// TwinCAT 3 PLC project LeakTesters
// ProgramVersion: 3.1.4024.0
// libraries:
//   Tc2_Standard, * (Beckhoff Automation GmbH)
//   Tc2_System, * (Beckhoff Automation GmbH)
//   Tc2_Utilities, * (Beckhoff Automation GmbH)
//   Tc3_EventLogger, * (Beckhoff Automation GmbH)
//   Tc3_Module, * (Beckhoff Automation GmbH)
//   VisuUserMgmt, * (System)
// project tree:
//   DUTs/ E_MachineState.TcDUT, E_StationState.TcDUT, ST_ActiveEventsHMI.TcDUT (not stored), ST_AlarmHistory.TcDUT (not stored), ST_Events.TcDUT, ST_Heightlimit.TcDUT, ST_MachineStatusStruct.TcDUT, ST_MasterControlStruct.TcDUT, ST_MeasureStatistics.TcDUT, ST_Nest.TcDUT, ST_PartsInspection.TcDUT, ST_StandardStationStruct.TcDUT, ST_UserLogHMI.TcDUT (not stored)
//   DUTs/IO/i28/ st_i28General_I_O.TcDUT (not stored), st_i28LasResult.TcDUT (not stored), st_i28LiveMeasurement.TcDUT (not stored)
//   DUTs/IO/ E_BoxDiag.TcDUT, E_BoxState.TcDUT, E_TerminalState.TcDUT, st_Box_Info.TcDUT, st_EL1809.TcDUT, st_EL2809.TcDUT, st_Terminal_Info.TcDUT
//   GVLs/ GVL_Constants.TcGVL, GVL_HMI_GLOBAL.TcGVL, GVL_IO.TcGVL, GVL_MASTER.TcGVL, GVL_PERSIST.TcGVL
//   / PlcTask.TcTTO
//   POUs/A_Master/ Main_Master.TcPOU, PRG_FaultHandling.TcPOU, PRG_MachineStatus.TcPOU, PRG_MasterCycle.TcPOU, PRG_MasterSystemTime.TcPOU, PRG_TerminBoxInfo.TcPOU
//   POUs/C_LeakTest/ PRG_Fault_LeakTest.TcPOU, PRG_LeakTest.TcPOU, PRG_LeakTestEvents_Info.TcPOU
//   POUs/E_HMI/ PRG_HMI.TcPOU
//   POUs/G_Utility/ FB_Alarms.TcPOU, FB_BoxInfo.TcPOU, FB_DayOfYear.TcPOU, FB_EventLog.TcPOU (not stored), FB_HeightMeasurement.TcPOU, FB_HeightTest.TcPOU, FB_Pulse.TcPOU (not stored), FB_TerminalInfo.TcPOU, FB_TimeControl.TcPOU (not stored), PRG_Puls.TcPOU
//   POUs/ MAIN.TcPOU
// real-time tasks:
//   TASK PlcTask: cycle T#10ms, priority 20, ADS port 350
// I/O:
//   DEVICE Device 1 (EtherCAT), AmsNetId 172.18.236.47.2.1
//     Term 9 (EK1100) [EK1100 EtherCAT Coupler (2A E-Bus)]
//       Term 10 (EL6070-0033) [EL6070-0033 1Ch. Licence key terminal, individual licences]
//       Term 11 (EL1809) [EL1809 16Ch. Dig. Input 24V, 3ms]
//       Term 12 (EL2809-0015) [EL2809-0015 16Ch. Dig. Output 24V DC, 0.35A, not short-circuit proof]
//       Term 13 (EL6631) [EL6631 PROFINET IO Controller]
//       Term 14 (EL9011) [EL9011 End Terminal]
//   DEVICE Device 2 (EL6631), AmsNetId 172.18.236.47.3.1
//     i28 [Cincinnati Test Systems 1-port Device 00210]
//       modules: Term 10 (DAP Module), Term 11 (PLC Input), Term 12 (PLC Output  )
// variable links:
//   LeakTesters/LeakTesters Instance <-> Device 1 (EtherCAT)/Term 9 (EK1100)/Term 11 (EL1809)
//     PlcTask Inputs/GVL_IO.dwTerminalInfo[3].nTerminal_State <-> InfoData/State
//     PlcTask Inputs/GVL_IO.dw_T02_EL1809.iCalmpClosed <-> Channel 1/Input
//     PlcTask Inputs/GVL_IO.dw_T02_EL1809.iPartPresent <-> Channel 2/Input
//   LeakTesters/LeakTesters Instance <-> Device 1 (EtherCAT)/Term 9 (EK1100)/Term 12 (EL2809-0015)
//     PlcTask Inputs/GVL_IO.dwTerminalInfo[4].nTerminal_State <-> InfoData/State
//     PlcTask Outputs/GVL_IO.dw_T03_EL2809.qEL2809_Ch3 <-> Channel 3/Output
//     PlcTask Outputs/GVL_IO.dw_T03_EL2809.qPassIndicatorGreen <-> Channel 1/Output
//     PlcTask Outputs/GVL_IO.dw_T03_EL2809.qRejectIndicatorRed <-> Channel 2/Output
//   LeakTesters/LeakTesters Instance <-> Device 1 (EtherCAT)/Term 9 (EK1100)/Term 13 (EL6631)
//     PlcTask Inputs/GVL_IO.dwTerminalInfo[5].nTerminal_State <-> InfoData/State
//   LeakTesters/LeakTesters Instance <-> Device 2 (EL6631)/i28
//     PlcTask Inputs/GVL_IO.dwBoxInfo[16].nPnIoBoxDiag <-> Inputs/PnIoBoxDiag
//     PlcTask Inputs/GVL_IO.dwBoxInfo[16].nPnIoBoxState <-> Inputs/PnIoBoxState
//     PlcTask Inputs/GVL_IO.dw_B07_i28General_I_O.bInput1 <-> API/Term 11 (PLC Input)/Subterm 15 (Instrument Status)/Inputs/Instrument Status/User_Configurable_Input_1
//     PlcTask Inputs/GVL_IO.dw_B07_i28General_I_O.bInput10 <-> API/Term 11 (PLC Input)/Subterm 15 (Instrument Status)/Inputs/Instrument Status/User_Configurable_Input_10
//     PlcTask Inputs/GVL_IO.dw_B07_i28General_I_O.bInput11 <-> API/Term 11 (PLC Input)/Subterm 15 (Instrument Status)/Inputs/Instrument Status/User_Configurable_Input_11
//     PlcTask Inputs/GVL_IO.dw_B07_i28General_I_O.bInput12 <-> API/Term 11 (PLC Input)/Subterm 15 (Instrument Status)/Inputs/Instrument Status/User_Configurable_Input_12
//     PlcTask Inputs/GVL_IO.dw_B07_i28General_I_O.bInput13 <-> API/Term 11 (PLC Input)/Subterm 15 (Instrument Status)/Inputs/Instrument Status/User_Configurable_Input_13
//     PlcTask Inputs/GVL_IO.dw_B07_i28General_I_O.bInput14 <-> API/Term 11 (PLC Input)/Subterm 15 (Instrument Status)/Inputs/Instrument Status/User_Configurable_Input_14
//     PlcTask Inputs/GVL_IO.dw_B07_i28General_I_O.bInput15 <-> API/Term 11 (PLC Input)/Subterm 15 (Instrument Status)/Inputs/Instrument Status/User_Configurable_Input_15
//     PlcTask Inputs/GVL_IO.dw_B07_i28General_I_O.bInput16 <-> API/Term 11 (PLC Input)/Subterm 15 (Instrument Status)/Inputs/Instrument Status/User_Configurable_Input_16
//     PlcTask Inputs/GVL_IO.dw_B07_i28General_I_O.bInput2 <-> API/Term 11 (PLC Input)/Subterm 15 (Instrument Status)/Inputs/Instrument Status/User_Configurable_Input_2
//     PlcTask Inputs/GVL_IO.dw_B07_i28General_I_O.bInput3 <-> API/Term 11 (PLC Input)/Subterm 15 (Instrument Status)/Inputs/Instrument Status/User_Configurable_Input_3
//     PlcTask Inputs/GVL_IO.dw_B07_i28General_I_O.bInput4 <-> API/Term 11 (PLC Input)/Subterm 15 (Instrument Status)/Inputs/Instrument Status/User_Configurable_Input_4
//     PlcTask Inputs/GVL_IO.dw_B07_i28General_I_O.bInput5 <-> API/Term 11 (PLC Input)/Subterm 15 (Instrument Status)/Inputs/Instrument Status/User_Configurable_Input_5
//     PlcTask Inputs/GVL_IO.dw_B07_i28General_I_O.bInput6 <-> API/Term 11 (PLC Input)/Subterm 15 (Instrument Status)/Inputs/Instrument Status/User_Configurable_Input_6
//     PlcTask Inputs/GVL_IO.dw_B07_i28General_I_O.bInput7 <-> API/Term 11 (PLC Input)/Subterm 15 (Instrument Status)/Inputs/Instrument Status/User_Configurable_Input_7
//     PlcTask Inputs/GVL_IO.dw_B07_i28General_I_O.bInput8 <-> API/Term 11 (PLC Input)/Subterm 15 (Instrument Status)/Inputs/Instrument Status/User_Configurable_Input_8
//     PlcTask Inputs/GVL_IO.dw_B07_i28General_I_O.bInput9 <-> API/Term 11 (PLC Input)/Subterm 15 (Instrument Status)/Inputs/Instrument Status/User_Configurable_Input_9
//     PlcTask Inputs/GVL_IO.dw_B07_i28General_I_O.bInstrumentReady <-> API/Term 11 (PLC Input)/Subterm 15 (Instrument Status)/Inputs/Instrument Status/Instrument_Ready
//     PlcTask Inputs/GVL_IO.dw_B07_i28General_I_O.bMalfunction <-> API/Term 11 (PLC Input)/Subterm 15 (Instrument Status)/Inputs/Instrument Status/Malfunction
//     PlcTask Inputs/GVL_IO.dw_B07_i28General_I_O.bProgramAccept <-> API/Term 11 (PLC Input)/Subterm 15 (Instrument Status)/Inputs/Instrument Status/Program_Accept
//     PlcTask Inputs/GVL_IO.dw_B07_i28General_I_O.bProgramReject <-> API/Term 11 (PLC Input)/Subterm 15 (Instrument Status)/Inputs/Instrument Status/Program_Reject
//     PlcTask Inputs/GVL_IO.dw_B07_i28General_I_O.bTestActiveLiveData <-> API/Term 11 (PLC Input)/Subterm 15 (Instrument Status)/Inputs/Instrument Status/Test_Active_Live_Data
//     PlcTask Inputs/GVL_IO.dw_B07_i28General_I_O.nCurrentProgramNumber <-> API/Term 11 (PLC Input)/Subterm 15 (Instrument Status)/Inputs/Current_Program Number
//     PlcTask Inputs/GVL_IO.dw_B07_i28LastResult.ibTestEvaluation0 <-> API/Term 11 (PLC Input)/Subterm 17 (Last test result)/Inputs/Test Evaluation Code/Test_Evaluation_Code_Bit_0
//     PlcTask Inputs/GVL_IO.dw_B07_i28LastResult.ibTestEvaluation1 <-> API/Term 11 (PLC Input)/Subterm 17 (Last test result)/Inputs/Test Evaluation Code/Test_Evaluation_Code_Bit_1
//     PlcTask Inputs/GVL_IO.dw_B07_i28LastResult.ibTestEvaluation2 <-> API/Term 11 (PLC Input)/Subterm 17 (Last test result)/Inputs/Test Evaluation Code/Test_Evaluation_Code_Bit_2
//     PlcTask Inputs/GVL_IO.dw_B07_i28LastResult.ibTestEvaluation3 <-> API/Term 11 (PLC Input)/Subterm 17 (Last test result)/Inputs/Test Evaluation Code/Test_Evaluation_Code_Bit_3
//     PlcTask Inputs/GVL_IO.dw_B07_i28LastResult.inChannelNumber <-> API/Term 11 (PLC Input)/Subterm 17 (Last test result)/Inputs/Channel Number
//     PlcTask Inputs/GVL_IO.dw_B07_i28LastResult.inMeasurement1 <-> API/Term 11 (PLC Input)/Subterm 17 (Last test result)/Inputs/Result Measurement 1
//     PlcTask Inputs/GVL_IO.dw_B07_i28LastResult.inMeasurement2 <-> API/Term 11 (PLC Input)/Subterm 17 (Last test result)/Inputs/Result Measurement 2
//     PlcTask Inputs/GVL_IO.dw_B07_i28LastResult.inPartEvaluation <-> API/Term 11 (PLC Input)/Subterm 17 (Last test result)/Inputs/Part Evaluation Code
//     PlcTask Inputs/GVL_IO.dw_B07_i28LastResult.inPrecisionCode <-> API/Term 11 (PLC Input)/Subterm 17 (Last test result)/Inputs/Precision Code
//     PlcTask Inputs/GVL_IO.dw_B07_i28LastResult.inProgramNumber <-> API/Term 11 (PLC Input)/Subterm 17 (Last test result)/Inputs/Program Number
//     PlcTask Inputs/GVL_IO.dw_B07_i28LastResult.inTestPort <-> API/Term 11 (PLC Input)/Subterm 17 (Last test result)/Inputs/Test Port
//     PlcTask Inputs/GVL_IO.dw_B07_i28LastResult.inTestType <-> API/Term 11 (PLC Input)/Subterm 17 (Last test result)/Inputs/Test Type Code
//     PlcTask Inputs/GVL_IO.dw_B07_i28LastResult.inUniqueID <-> API/Term 11 (PLC Input)/Subterm 17 (Last test result)/Inputs/Unique ID
//     PlcTask Inputs/GVL_IO.dw_B07_i28LastResult.inUnitCode1 <-> API/Term 11 (PLC Input)/Subterm 17 (Last test result)/Inputs/Unit Code[0]
//     PlcTask Inputs/GVL_IO.dw_B07_i28LastResult.inUnitCode2 <-> API/Term 11 (PLC Input)/Subterm 17 (Last test result)/Inputs/Unit Code[1]
//     PlcTask Inputs/GVL_IO.dw_B07_i28LastResult.inVariableCode1 <-> API/Term 11 (PLC Input)/Subterm 17 (Last test result)/Inputs/Variable Code[0]
//     PlcTask Inputs/GVL_IO.dw_B07_i28LastResult.inVariableCode2 <-> API/Term 11 (PLC Input)/Subterm 17 (Last test result)/Inputs/Variable Code[1]
//     PlcTask Inputs/GVL_IO.dw_B07_i28LiveMeasurement.inCurrentProgramNumber <-> API/Term 11 (PLC Input)/Subterm 16 (Live Measurement Data)/Inputs/Current Program Number
//     PlcTask Inputs/GVL_IO.dw_B07_i28LiveMeasurement.inMeasurement1 <-> API/Term 11 (PLC Input)/Subterm 16 (Live Measurement Data)/Inputs/Measurement 1 (Timer)
//     PlcTask Inputs/GVL_IO.dw_B07_i28LiveMeasurement.inMeasurement2 <-> API/Term 11 (PLC Input)/Subterm 16 (Live Measurement Data)/Inputs/Measurement 2 (Pressure)
//     PlcTask Inputs/GVL_IO.dw_B07_i28LiveMeasurement.inMeasurement3 <-> API/Term 11 (PLC Input)/Subterm 16 (Live Measurement Data)/Inputs/Measurement 3 (Pressure Loss/Rate)
//     PlcTask Inputs/GVL_IO.dw_B07_i28LiveMeasurement.inMeasurement4 <-> API/Term 11 (PLC Input)/Subterm 16 (Live Measurement Data)/Inputs/Measurement 4 (Flow/Leak)
//     PlcTask Inputs/GVL_IO.dw_B07_i28LiveMeasurement.inPrecisionCode1 <-> API/Term 11 (PLC Input)/Subterm 16 (Live Measurement Data)/Inputs/Precision Code[0]
//     PlcTask Inputs/GVL_IO.dw_B07_i28LiveMeasurement.inPrecisionCode2 <-> API/Term 11 (PLC Input)/Subterm 16 (Live Measurement Data)/Inputs/Precision Code[1]
//     PlcTask Inputs/GVL_IO.dw_B07_i28LiveMeasurement.inPrecisionCode3 <-> API/Term 11 (PLC Input)/Subterm 16 (Live Measurement Data)/Inputs/Precision Code[2]
//     PlcTask Inputs/GVL_IO.dw_B07_i28LiveMeasurement.inPrecisionCode4 <-> API/Term 11 (PLC Input)/Subterm 16 (Live Measurement Data)/Inputs/Precision Code[3]
//     PlcTask Inputs/GVL_IO.dw_B07_i28LiveMeasurement.inSegmentCode <-> API/Term 11 (PLC Input)/Subterm 16 (Live Measurement Data)/Inputs/Segment Code
//     PlcTask Inputs/GVL_IO.dw_B07_i28LiveMeasurement.inUniqueID <-> API/Term 11 (PLC Input)/Subterm 16 (Live Measurement Data)/Inputs/Unique ID
//     PlcTask Inputs/GVL_IO.dw_B07_i28LiveMeasurement.inUnitCode1 <-> API/Term 11 (PLC Input)/Subterm 16 (Live Measurement Data)/Inputs/Unit Code[0]
//     PlcTask Inputs/GVL_IO.dw_B07_i28LiveMeasurement.inUnitCode2 <-> API/Term 11 (PLC Input)/Subterm 16 (Live Measurement Data)/Inputs/Unit Code[1]
//     PlcTask Inputs/GVL_IO.dw_B07_i28LiveMeasurement.inUnitCode3 <-> API/Term 11 (PLC Input)/Subterm 16 (Live Measurement Data)/Inputs/Unit Code[2]
//     PlcTask Inputs/GVL_IO.dw_B07_i28LiveMeasurement.inUnitCode4 <-> API/Term 11 (PLC Input)/Subterm 16 (Live Measurement Data)/Inputs/Unit Code[3]
//     PlcTask Inputs/GVL_IO.dw_B07_i28LiveMeasurement.inVariableCode1 <-> API/Term 11 (PLC Input)/Subterm 16 (Live Measurement Data)/Inputs/Variable Code[0]
//     PlcTask Inputs/GVL_IO.dw_B07_i28LiveMeasurement.inVariableCode2 <-> API/Term 11 (PLC Input)/Subterm 16 (Live Measurement Data)/Inputs/Variable Code[1]
//     PlcTask Inputs/GVL_IO.dw_B07_i28LiveMeasurement.inVariableCode3 <-> API/Term 11 (PLC Input)/Subterm 16 (Live Measurement Data)/Inputs/Variable Code[2]
//     PlcTask Inputs/GVL_IO.dw_B07_i28LiveMeasurement.inVariableCode4 <-> API/Term 11 (PLC Input)/Subterm 16 (Live Measurement Data)/Inputs/Variable Code[3]
//     PlcTask Outputs/GVL_IO.dw_B07_i28General_I_O.bChangeProgram <-> API/Term 12 (PLC Output  )/Subterm 18 (Instrument Control )/Outputs/Instrument Control/Change_Program
//     PlcTask Outputs/GVL_IO.dw_B07_i28General_I_O.bOutput1 <-> API/Term 12 (PLC Output  )/Subterm 18 (Instrument Control )/Outputs/Instrument Control/User_Configurable_Output_1
//     PlcTask Outputs/GVL_IO.dw_B07_i28General_I_O.bOutput10 <-> API/Term 12 (PLC Output  )/Subterm 18 (Instrument Control )/Outputs/Instrument Control/User_Configurable_Output_10
//     PlcTask Outputs/GVL_IO.dw_B07_i28General_I_O.bOutput11 <-> API/Term 12 (PLC Output  )/Subterm 18 (Instrument Control )/Outputs/Instrument Control/User_Configurable_Output_11
//     PlcTask Outputs/GVL_IO.dw_B07_i28General_I_O.bOutput12 <-> API/Term 12 (PLC Output  )/Subterm 18 (Instrument Control )/Outputs/Instrument Control/User_Configurable_Output_12
//     PlcTask Outputs/GVL_IO.dw_B07_i28General_I_O.bOutput13 <-> API/Term 12 (PLC Output  )/Subterm 18 (Instrument Control )/Outputs/Instrument Control/User_Configurable_Output_13
//     PlcTask Outputs/GVL_IO.dw_B07_i28General_I_O.bOutput14 <-> API/Term 12 (PLC Output  )/Subterm 18 (Instrument Control )/Outputs/Instrument Control/User_Configurable_Output_14
//     PlcTask Outputs/GVL_IO.dw_B07_i28General_I_O.bOutput15 <-> API/Term 12 (PLC Output  )/Subterm 18 (Instrument Control )/Outputs/Instrument Control/User_Configurable_Output_15
//     PlcTask Outputs/GVL_IO.dw_B07_i28General_I_O.bOutput16 <-> API/Term 12 (PLC Output  )/Subterm 18 (Instrument Control )/Outputs/Instrument Control/User_Configurable_Output_16
//     PlcTask Outputs/GVL_IO.dw_B07_i28General_I_O.bOutput2 <-> API/Term 12 (PLC Output  )/Subterm 18 (Instrument Control )/Outputs/Instrument Control/User_Configurable_Output_2
//     PlcTask Outputs/GVL_IO.dw_B07_i28General_I_O.bOutput3 <-> API/Term 12 (PLC Output  )/Subterm 18 (Instrument Control )/Outputs/Instrument Control/User_Configurable_Output_3
//     PlcTask Outputs/GVL_IO.dw_B07_i28General_I_O.bOutput4 <-> API/Term 12 (PLC Output  )/Subterm 18 (Instrument Control )/Outputs/Instrument Control/User_Configurable_Output_4
//     PlcTask Outputs/GVL_IO.dw_B07_i28General_I_O.bOutput5 <-> API/Term 12 (PLC Output  )/Subterm 18 (Instrument Control )/Outputs/Instrument Control/User_Configurable_Output_5
//     PlcTask Outputs/GVL_IO.dw_B07_i28General_I_O.bOutput6 <-> API/Term 12 (PLC Output  )/Subterm 18 (Instrument Control )/Outputs/Instrument Control/User_Configurable_Output_6
//     PlcTask Outputs/GVL_IO.dw_B07_i28General_I_O.bOutput7 <-> API/Term 12 (PLC Output  )/Subterm 18 (Instrument Control )/Outputs/Instrument Control/User_Configurable_Output_7
//     PlcTask Outputs/GVL_IO.dw_B07_i28General_I_O.bOutput8 <-> API/Term 12 (PLC Output  )/Subterm 18 (Instrument Control )/Outputs/Instrument Control/User_Configurable_Output_8
//     PlcTask Outputs/GVL_IO.dw_B07_i28General_I_O.bOutput9 <-> API/Term 12 (PLC Output  )/Subterm 18 (Instrument Control )/Outputs/Instrument Control/User_Configurable_Output_9
//     PlcTask Outputs/GVL_IO.dw_B07_i28General_I_O.bReset <-> API/Term 12 (PLC Output  )/Subterm 18 (Instrument Control )/Outputs/Instrument Control/Reset
//     PlcTask Outputs/GVL_IO.dw_B07_i28General_I_O.bSetProgram[0] <-> API/Term 12 (PLC Output  )/Subterm 18 (Instrument Control )/Outputs/Desired Program Number[0]
//     PlcTask Outputs/GVL_IO.dw_B07_i28General_I_O.bSetProgram[1] <-> API/Term 12 (PLC Output  )/Subterm 18 (Instrument Control )/Outputs/Desired Program Number[1]
//     PlcTask Outputs/GVL_IO.dw_B07_i28General_I_O.bSetProgram[2] <-> API/Term 12 (PLC Output  )/Subterm 18 (Instrument Control )/Outputs/Desired Program Number[2]
//     PlcTask Outputs/GVL_IO.dw_B07_i28General_I_O.bSetProgram[3] <-> API/Term 12 (PLC Output  )/Subterm 18 (Instrument Control )/Outputs/Desired Program Number[3]
//     PlcTask Outputs/GVL_IO.dw_B07_i28General_I_O.bSetProgram[4] <-> API/Term 12 (PLC Output  )/Subterm 18 (Instrument Control )/Outputs/Desired Program Number[4]
//     PlcTask Outputs/GVL_IO.dw_B07_i28General_I_O.bSetProgram[5] <-> API/Term 12 (PLC Output  )/Subterm 18 (Instrument Control )/Outputs/Desired Program Number[5]
//     PlcTask Outputs/GVL_IO.dw_B07_i28General_I_O.bSetProgram[6] <-> API/Term 12 (PLC Output  )/Subterm 18 (Instrument Control )/Outputs/Desired Program Number[6]
//     PlcTask Outputs/GVL_IO.dw_B07_i28General_I_O.bSetProgram[7] <-> API/Term 12 (PLC Output  )/Subterm 18 (Instrument Control )/Outputs/Desired Program Number[7]
//     PlcTask Outputs/GVL_IO.dw_B07_i28General_I_O.bStart <-> API/Term 12 (PLC Output  )/Subterm 18 (Instrument Control )/Outputs/Instrument Control/Start
//     PlcTask Outputs/GVL_IO.dw_B07_i28General_I_O.bStop <-> API/Term 12 (PLC Output  )/Subterm 18 (Instrument Control )/Outputs/Instrument Control/Stop
//     PlcTask Outputs/GVL_IO.dw_B07_i28General_I_O.bVentHalt <-> API/Term 12 (PLC Output  )/Subterm 18 (Instrument Control )/Outputs/Instrument Control/Vent_Halt

CONFIGURATION LeakTesters
    RESOURCE PLC ON TwinCAT3
        TASK PlcTask(INTERVAL := T#10ms, PRIORITY := 20);
        PROGRAM MAIN WITH PlcTask : MAIN;
    END_RESOURCE
END_CONFIGURATION

// ---- DUTs/E_MachineState.TcDUT
{attribute 'qualified_only'}
{attribute 'strict'}
TYPE E_MachineState :
(
	SYSTEM_POWER_UP:=0,
	IMMEDIATE_STOPPED:=100,
	SYSTEM_INITIALISING:=110,
	SYSTEM_READY_TO_START:=120,
	SYSTEM_AUTO_CYCLE:=130,
	SYSTEM_DWELL:=140,
	STOPPING:=145,
	CYCLE_STOPPED:=150,
	MANUAL_MODE:=160 ,
	MAINTENANCE_MODE:=165,
	IMMEDIATE_FAULT:=170,
	CYCLE_STOP_FAULT:=180
);
END_TYPE

// ---- DUTs/E_StationState.TcDUT
{attribute 'qualified_only'}
{attribute 'strict'}
TYPE E_StationState :
(
	RESETTING := 0,
	PRE_ELIMINARY_CHECKS,
	TRY_HOMING,
	HOMING,
	HOMING_DONE,
	READY,
	STARTING,
	DWELL,
	OPERATING,
	
//VALUES FOR UCB
	
//standard steps
	ERROR,
	COMPLETE
);
END_TYPE

// ---- DUTs/IO/E_BoxDiag.TcDUT
{attribute 'qualified_only'}
{attribute 'strict'}
TYPE E_BoxDiag :
(
	No_diagnosis                                   :=0,
    IOC_AR_is_not_established                      := 1,
    IOC_AR_is_established                          := 2,
    IOC_AR_is_established_but_no_application_ready := 4,
    IOC_AR_is_established_but_module_difference    := 8,
    At_least_one_AlarmCR_got_a_diagnosis_alarm     := 10,
    At_least_one_InputCR_is_invalid                := 100,
    At_least_one_InputCR_Provider_is_in_stop       := 200,
    At_least_one_InputCR_Problemindicator_is_set   := 400,
    At_least_one_OutputCR_is_invalid               := 1000,
    At_least_one_OutputCR_Provider_is_in_stop      := 2000,
    At_least_one_OutputCR_Problemindicator_is_set  := 4000
);
END_TYPE

// ---- DUTs/IO/E_BoxState.TcDUT
{attribute 'qualified_only'}
{attribute 'strict'}
TYPE E_BoxState :
(
	No_error                                                                     := 0,
    Profinet_device_state_machine_is_in_boot_mode                                := 1,
    Device_NOT_found                                                             := 2,
    The_stationname_is_not_unique                                                := 3,
    IP_could_not_be_set                                                          := 4,
    IP_conflict                                                                  := 5,
    DCP_set_was_not_successful                                                   := 6,
    Watchdog_error                                                               := 7,
    Datahold_error                                                               := 8,
    RTC3_Sync_mode_could_NOT_be_initiated                                        := 9,
    Profinet_controller_has_a_link_error                                         := 10,
    The_aliasname_is_not_unique                                                  := 11,
    The_automatic_name_assignement_isnt_possible_wrong_device_type               := 12,
    IOC_AR_is_established_but_no_application_ready                               := 13,
    IOC_AR_is_established_but_module_difference                                  := 14,
    At_least_one_InputCR_is_invalid_provider_in_stop_OR_problemindicator_is_set  := 15,
    At_least_one_OutputCR_is_invalid_provider_in_stop_OR_problemindicator_is_set := 16,
    Only_for_EtherCAT_gateways_WC_State_OF_cyclic_EtherCAT_frame_is_1            := 31
);
END_TYPE

// ---- DUTs/IO/E_TerminalState.TcDUT
{attribute 'qualified_only'}
{attribute 'strict'}
TYPE E_TerminalState :
(
	 INIT   := 0 ,
     PREOP  := 2 ,
     BOOT   := 3 ,
     SAFEOP := 4 ,
     OP     := 8 

);
END_TYPE

// ---- DUTs/IO/st_Box_Info.TcDUT
TYPE st_Box_Info :
STRUCT
	nPnIoBoxState    AT%I* : UINT;
    nPnIoBoxDiag     AT%I* : UINT;
    eBoxState              : E_BoxState;
	eBoxDiag               : E_BoxDiag;
	fbBoxInfo              : FB_BoxInfo;
	sBoxState              : STRING;
	sBoxDiag               : STRING;
	
END_STRUCT
END_TYPE

// ---- DUTs/IO/st_EL1809.TcDUT
TYPE st_EL1809 :
STRUCT
	
		//--------------------------------------------------------------------------------------------------------
	sTerminalName                                           :   STRING(200):= 'EL1809 | 16-Channel Digital Input';
    //============================================================================================================================	
	// TERMINAL - EL1809 16-Channel Digital Input Terminal 
    (*Terminal 02*)
	iCalmpClosed                			AT %I*			: 	BOOL;	// EL1809 channel 1
	iPartPresent                            AT %I*			: 	BOOL;	// EL1809 channel 2
	iEL1809_Ch3								AT %I*	 		: 	BOOL;	// EL1809 channel 3
	iEL1809_Ch4								AT %I*	 		: 	BOOL;	// EL1809 channel 4
	iEL1809_Ch5	    		                AT %I*	 		: 	BOOL;	// EL1809 channel 5 		     			
	iEL1809_Ch6			  					AT %I*			: 	BOOL;	// EL1809 channel 6
	iEL1809_Ch7		    					AT %I*	 		: 	BOOL;	// EL1809 channel 7 
	iEL1809_Ch8			   					AT %I*	 		: 	BOOL;	// EL1809 channel 8 
    iEL1809_Ch9			                    AT %I*	 		: 	BOOL;	// EL1809 channel 9 
	iEL1809_Ch10			                AT %I*          :   BOOL;   // EL1809 channel 10 
	iEL1809_Ch11		                    AT %I*          :   BOOL;   // EL1809 channel 11
	iEL1809_Ch12		                    AT %I*          :   BOOL;   // EL1809 channel 12	   
	iEL1809_Ch13			   		    	AT %I*	 		: 	BOOL;	// EL1809 channel 13   
	iEL1809_Ch14							AT %I*	 		: 	BOOL;	// EL1809 channel 14 
	iEL1809_Ch15	  						AT %I*			: 	BOOL;	// EL1809 channel 15  
	iEL1809_Ch16							AT %I*	 		: 	BOOL;	// EL1809 channel 16  

END_STRUCT
END_TYPE

// ---- DUTs/IO/st_EL2809.TcDUT
TYPE st_EL2809 :
STRUCT
	
		sTerminalName                                           :   STRING(200):= 'EL2809 | 16-Channel Digital Output';
	//=============================================================================================================
	// TERMINAL - EL2809	16-Channel Digital Output Terminal	 (Term ...)
	qPassIndicatorGreen 					AT %Q*			: 	BOOL;	// EL2809 channel 1
	qRejectIndicatorRed						AT %Q* 			: 	BOOL;	// EL2809 channel 2
	qEL2809_Ch3				                AT %Q*          :   BOOL;   // EL2809 channel 3
	qEL2809_Ch4				            	AT %Q*          :   BOOL;   // EL2809 channel 4   	
	qEL2809_Ch5		     					AT %Q*	 		: 	BOOL;	// EL2809 channel 5	
	qEL2809_Ch6	    		            	AT %Q*	 		: 	BOOL;	// EL2809 channel 6	
    qEL2809_Ch7	                        	AT %Q*          :   BOOL;   // EL2809 channel 7	
	qEL2809_Ch8								AT %Q*	 		: 	BOOL;	// EL2809 channel 8 
	qEL2809_Ch9				                AT %Q*          :   BOOL;   // EL2809 channel 9
	qEL2809_Ch10				            AT %Q*          :   BOOL;   // EL2809 channel 10   	
	qEL2809_Ch11		     				AT %Q*	 		: 	BOOL;	// EL2809 channel 11	
	qEL2809_Ch12	    		            AT %Q*	 		: 	BOOL;	// EL2809 channel 12	
    qEL2809_Ch13	                        AT %Q*          :   BOOL;   // EL2809 channel 13	
	qEL2809_Ch14							AT %Q*	 		: 	BOOL;	// EL2809 channel 14 
    qEL2809_Ch15        			        AT %Q*	 		: 	BOOL;	// EL2809 channel 15 
	qEL2809_Ch16                            AT %Q*	 		: 	BOOL;	// EL2809 channel 16 
	
	
END_STRUCT
END_TYPE

// ---- DUTs/IO/st_Terminal_Info.TcDUT
TYPE st_Terminal_Info :
STRUCT
	nTerminal_State                        AT %I*			:    UINT;	// Terminal State from IO Terminal Info Data
    eTerminal_State                                         :    E_TerminalState;
	sTerminalInfo                                           :    STRING;
    fbTerminalInfo                                          :    FB_TerminalInfo;
END_STRUCT
END_TYPE

// ---- DUTs/ST_Events.TcDUT
TYPE ST_Events :
STRUCT
	bImmediateFault				:BOOL;
	bCycleStopFault				:BOOL;
	bCycleStopRequest			:BOOL;

	bEventTextsSet				:BOOL; //True after event texts are set 
	aEventFlags					:ARRAY[0..127] OF BOOL;
	aEventTimers				:ARRAY[0..127] OF TON;
	aEventTexts					:ARRAY[0..127] OF T_MaxString;
END_STRUCT
END_TYPE

// ---- DUTs/ST_Heightlimit.TcDUT
TYPE ST_Heightlimit :
STRUCT
	LOW:   INT;
	HIGH:  INT;
	
END_STRUCT
END_TYPE

// ---- DUTs/ST_MachineStatusStruct.TcDUT
TYPE ST_MachineStatusStruct :
STRUCT
	nState						: INT;
	//nStateBuffer				: INT;
	eMachineState				:E_MachineState;	
	bSystemPowerUp 				:BOOL;
	bImmediateStopped 			:BOOL;
	bSystemInitialising 		:BOOL;
	bSystemReadyToStart 		:BOOL;
	bSystemAutoCycle 			:BOOL;
	bSystemDwell 				:BOOL;
	bSystemStopping				:BOOL;	
	bCycleStopped 				:BOOL;
	bImmediateFault 			:BOOL;
	bCycleStopFault 			:BOOL;
	bManualMode					:BOOL;
    bSystemStandby              :BOOL;		
	
	sMachineStatusText			:STRING;
	nMachineStatusTxtCol		:DWORD;
	nMachineStatusColour		:DWORD;
	sBannerTextColor			:STRING ;
	sBannerBckColor				:STRING ;
END_STRUCT
END_TYPE

// ---- DUTs/ST_MasterControlStruct.TcDUT
TYPE ST_MasterControlStruct :
STRUCT
	bAbort									:BOOL;
	bNoMachineImmediateFault				:BOOL;
	bNoStationImmediateFault				:BOOL;
	bNoCycleStopFault						:BOOL;
	bAllStationsHomed						:BOOL;
	bAllStationsCycledStopped				:BOOL;
	bCycleStopRequest						:BOOL;
	bDwellRequest							:BOOL;
	bManualModeRequest						:BOOL;
	bFreezeMachineStatus					:BOOL;
	bPowerUpTimerComplete					:BOOL;
	bSystemInitialisingTimerComplete		:BOOL;
	bSystemInitialisingTimeoutComplete		:BOOL;
	bResetImmediateFaultDelay				:BOOL;
	
	bAllStationsSafeToIndex					:BOOL;
	bAllStationsOKToIndex					:BOOL;
	bAllStationsNotMoving					:BOOL;
	
	bLineClearanceRequest					:BOOL;
	bLineClearanceComplete					:BOOL;
END_STRUCT
END_TYPE

// ---- DUTs/ST_MeasureStatistics.TcDUT
TYPE ST_MeasureStatistics :
STRUCT
	 bOutLimitMax	 : BOOL;
	 bOutLimitMin    : BOOL;
	 nMesureFaultMin : UINT;
	 nMesureFaultMax : UINT;
END_STRUCT
END_TYPE

// ---- DUTs/ST_Nest.TcDUT
TYPE ST_Nest :
STRUCT
		 

	 
     bNestPartProced    : BOOL;
	 bNestPresent       : BOOL;
	 
	 bPiecePass			: BOOL;
	 bPieceReject		: BOOL;
	 bLeakPass			: BOOL;
	 bLeakReject		: BOOL;
	 
	 
	 sLeakHMI			: WSTRING;
	 sPieceHMI			: WSTRING;

	 
	 sDate				: STRING;
	 sTime				: STRING;

END_STRUCT
END_TYPE

// ---- DUTs/ST_PartsInspection.TcDUT
TYPE ST_PartsInspection :
STRUCT
	
	nPartsGood						: DINT;
	nTotalPartsGood					: DINT;
	nPartsFailed					: DINT;
	nTotalPartsFailed				: DINT;					
	
	bPartok							: BOOL;
	bPartFail						: BOOL;
END_STRUCT
END_TYPE

// ---- DUTs/ST_StandardStationStruct.TcDUT
TYPE ST_StandardStationStruct :
STRUCT
	
		// Station Manager => Master Control
	nState 							: 	DINT := 100;//Station Cycle State
	bStationWaitOnInit              :   BOOL;       //Station Waiting For Initialisation Request
	bStationWaitOnRequest			:	BOOL;		//Station In Valide State Avaiting For Request Command
	bStationInProgress				: 	BOOL;		//Station In Progress With Cycle
	bStationInProgressInit          :   BOOL;       //Station In Progress With Imotialisation     
	bStationComplete				: 	BOOL;		//Station Complete Cycle - Flag Set After Every Cycle Finsh
	bStationCycleStopped			: 	BOOL;
	bStationHomed					: 	BOOL;		//Station Homed - All Station Functions Are Homed 
	bStationDone					:	BOOL;		//Sequence Finished With Success - Flag Set For One PLC Cycle
	bStationNotMoving				: 	BOOL;		//Station Parts Are Not Moving
	bStationInDwell					: 	BOOL;		//Station Waiting For External Action By Operator
	bStationAcknowledge             :   BOOL;       //Station Acknowledge request from Master 
	bStationInitDone                :   BOOL;       //Station Initialisation Progress Done
	// Master Control => Station Manager
	bStationInitRequest             :   BOOL;       //Request Commnad To Start Station Initialisation
	bStationRequest					: 	BOOL;		//Request Commnad To Start Station Cycle
	bStationCompleteAck				: 	BOOL;		//Request Commnad To Start Station Cycle
	bStationHomingRequest			:	BOOL;		//Staion Homing Requested By Manager Or Internal Functions
	bStationAbort					: 	BOOL;		//Station Abort By Manager
	bNoCycleStopRequest				:	BOOL;		//Stop Cycle Requested By Manager
	bNoCycleStopFault				: 	BOOL;		//No  Stop Fault On Station - Immidiat STOP Station
	bNoImmediateFault				: 	BOOL;		//No Immediate Fault On Station - Immidiat STOP Machine
	
	
	bStationManualRequestHMI		:	BOOL;		//Sequence Cycle Requested From HMI
	bStationInManualMode			:	BOOL;		//Station Sequence Manage By Operator

	bStationInStandByMode			:	BOOL;		//Sequence In Stand By State
	bStationFreezedByManager		: 	BOOL;		//Sequence Cycle Freezed (Suspend)  By Manager
	
	eStationState					: 	E_StationState; // state of sequence
	
	bPartOK							:	BOOL;		// 1-Cycle succeed
	bPartReject                     :   BOOL;       // 1-Cycle failed

	
	bStationWaiting                 :   BOOL; // Station in the  positiont waiting for work done
	bStationCycleCondition          :   BOOL; // Station in cycle move
END_STRUCT
END_TYPE

// ---- GVLs/GVL_Constants.TcGVL
VAR_GLOBAL CONSTANT
	sWHITE                              :   STRING(40)  := '{"color":"rgba(255,255,255,255)"}';
    sBLACK                              :   STRING(40)  := '{"color":"rgba(0,0,0,1)"}';
    sYELLOW                             :   STRING(40)  := '{"color":"rgba(255,255,0,1)"}';
    sGREEN                             	:   STRING(40)  := '{"color":"rgba(70,166,63,1)"}';
	sLGREEN                             :   STRING(40)  := '{"color":"rgba(58,211,20,1)"}';
    sORANGE                             :   STRING(40)  := '{"color":"rgba(255,153,51,1)"}';
    sNYPROORANGE                        :   STRING(40)  := '{"color":"rgba(255,140,0,1)"}';
    sRED                                :   STRING(40)  := '{"color":"rgba(255,0,0,1)"}';
	sLRED                               :   STRING(40)  := '{"color":"rgba(233,53,44,1)"}';
    sBLUE                               :   STRING(40)  := '{"color":"rgba(0,0,255,1)"}';
	sLBLUE                              :   STRING(40)  := '{"color":"rgba(0,162,232,1)"}';
    sGREY                               :   STRING(40)  := '{"color":"rgba(164,158,158,1)"}';
    sScreenGREY                         :   STRING(40)  := '{"color":"rgba(225,225,225,1)"}';
    sDARKGREY                           :   STRING(40)  := '{"color":"rgba(50,50,50,1)"}';
    sPURPLE                             :   STRING(40)  := '{"color":"rgba(128,0,128,1)"}';
    sVIOLET                             :   STRING(40)  := '{"color":"rgba(204,153,255,1)"}';
    sTRANSP                             :   STRING(40)  := '{"color":"rgba(255,255,255,0)"}';
    sGREENPass                          :   STRING(40)  := '{"color":"rgba(0,153,51,1)"}';
    sREDFail                            :   STRING(40)  := '{"color":"rgba(244,68,68,255)"}';
    sBLUEInProgress                     :   STRING(40)  := '{"color":"rgba(54,100,221,1)"}';
	sGREENISHTEAColor					:	STRING(40)  := '{"color":"rgba(60,192,134,255)"}'	;		

	nBLACK								: 	DWORD 	:= 	16#FF000000;	 // format: TTRRGGBB where T -> 00 = full transparency and FF = full opaque
	nWHITE								: 	DWORD 	:= 	16#FFFFFFFF;
	nYELLOW								: 	DWORD 	:= 	16#FFFFFF00; 
	nGREEN								: 	DWORD 	:= 	16#FF008A00;
	nLIGHTGREEN                         :   DWORD   :=  16#FF98FB89;
	nORANGE								: 	DWORD 	:= 	16#FFFFA500;
	nNYPROORANGE						:	DWORD	:=	16#FFF05322;//F05322;
	nRED								: 	DWORD 	:= 	16#FFFF0000;
	nBLUE								: 	DWORD 	:= 	16#FF0000FF;
	nLIGHTBLUE                          :   DWORD   :=  16#FF08ADF4;//FF9FDDFB;
	nGREY								: 	DWORD 	:= 	16#FFA9A9A9;	
	nDARKGREY							:	DWORD	:=	16#FF808080;
	nPURPLE								:	DWORD	:=	16#FF800080;
	nVIOLET								:	DWORD	:=	16#FFEE82EE;
	nTRANSP								:	DWORD	:=	16#00FFFFFF;	// full transparent WHITE
	
	nLCColNormal						:	DWORD	:= 16#10008A00;		// light curtain green
	nLCColBroken						:	DWORD	:= 16#64FF0000;		// light curtain red
END_VAR

// ---- GVLs/GVL_HMI_GLOBAL.TcGVL
{attribute 'qualified_only'}
VAR_GLOBAL
	
	//User Log, Shut down, Quit HMI
	bQuitHmi						: BOOL;
	sUserGroup						: STRING;
	sUserGroup2						: STRING;
	sUserName						: STRING;
	bLogOut							: BOOL;
	bUserLogedIntSignal				: BOOL;
	bShutDown						: BOOL;
	
	
	
	
	
	//General
	bStopButton						: BOOL;
	bStartButton					: BOOL;
	bResetButton					: BOOL;
	nRegionMain						: INT;
	bTrigerCamMan					: BOOL;
	bResetGoodParts					: BOOL;
	bResetFailedParts				: BOOL;
	bManualModeOff					: ARRAY[1..2] OF BOOL;
	
	aEventTexts						: ARRAY [0..767] OF T_MaxSTring; //Event texts - set only once
	bEventTextsSet					: BOOL;
	aEventFlags						: ARRAY [0..767] OF BOOL;		//All event states combined from master na stations
	aActiveEvents					: ARRAY [0..39] OF T_MaxSTring;	//Active events - connected to Alarm scree in HMI	
	stActiveEventsHMI				: ARRAY [0..39] OF ST_ActiveEventsHMI;
	
	aStatistics						: ARRAY [1..201] OF ST_Nest; // **LA 04092025 >> : ARRAY [1..200] OF ST_Nest;
	sMessageToOperator				: WSTRING(200);
	sActualProcess					: WSTRING(200);
	aIOScreen						: ARRAY [0..8] OF STRING(200);
	aManualScreen					: ARRAY [0..2] OF STRING(200);
	bResetPassAndFail				: BOOL;
	bEnableManualMode				: BOOL;
	bRejectPieceAcknowledge			: BOOL;
	bRejectPieceDialogTrig			: BOOL;
	bAutoCycleFaultDialog			: BOOL;
	bStopperPressEnable				: BOOL;
	nGeneralCycTime					: DINT;
		
	
	// ------ Screen Info / Data -----------	
	sSystemDate					: STRING;
	sSystemTime					: STRING;
	ntAMSNetID					: T_AmsNetId := '172.18.236.47.1.1';
	sStopperEnableDisable		:STRING(30); 
	
	
	//Leak Tester
	bLeakTestPass					: BOOL;
	uSetLeakProgramID				: USINT;
	bSetLeakProgramID				: BOOL;
	bResetLeakMan					: BOOL;
	bStartLeakMan					: BOOL;
	bStopLeakMan					: BOOL;
	bLoadLeakProg					: BOOL;
	uNewLeakProgID					: USINT;
		
	bResetLeakGoodParts				: BOOL;
	bResetLeakBadParts				: BOOL;
	nLeakTestCycTime				: DINT;	

END_VAR
VAR_GLOBAL PERSISTENT
	stAlarmHistory				:ARRAY [00..250] OF ST_AlarmHistory;
	aEventLog					:ARRAY [0..250] OF T_MaxSTring;	//Event log - connected to alarm history in HMI	
	aTimeLog					:ARRAY [0..250] OF T_MaxSTring;
	aDateLog					:ARRAY [0..250] OF T_MaxSTring;			
END_VAR

// ---- GVLs/GVL_IO.TcGVL
{attribute 'qualified_only'}
VAR_GLOBAL
	
    //--------------------------------------------------------------------------------------------------------

    dwTerminalInfo                                          : ARRAY[0..20] OF  st_Terminal_Info; // all terminal's status information 
	dwBoxInfo                                               : ARRAY[15..17] OF st_Box_Info;//Camera, Leak, Height
	//--------------------------------------------------------------------------------------------------------
	
	(* Terminal *)
	
	//	dw_T01_EK1100                                                	| EtherCAT Coupler 
	//	dw_T02_EL6070-0033                                           	| EtherCAT Terminal, license key for TwinCAT 3.1
	
	dw_T02_EL1809                                                		: st_EL1809; //16 Channel Digital Input ( 24VDC ) 
	dw_T03_EL2809                                                		: st_EL2809; // 16 Channel Digital Output ( 24VDC )
	//dw_T04_EL6631                                                	| EtherCAT Terminal, 2-port communication interface, PROFINET RT, controller - Data for Box's MDU1020 and SR2000W
 	//  dw_T05_EL9011                                                	| Bus end cover for E-bus contacts
	
	dw_B07_i28General_I_O												: st_i28General_I_O;
	dw_B07_i28LastResult												: st_i28LasResult;
	dw_B07_i28LiveMeasurement											: st_i28LiveMeasurement;
	
	
	
END_VAR

// ---- GVLs/GVL_MASTER.TcGVL
{attribute 'qualified_only'}
VAR_GLOBAL
	(*-----------------------------------------------------------------------------------------------------------------*)
	// System Pulses 
	bFlash1Hz						: BOOL;
	bFlash2Hz						: BOOL;
	bFlash4Hz				   		: BOOL;
	bFlash10Hz						: BOOL;
	bFlash10BHz        		  		: BOOL;
	bFlash100Hz      	      		: BOOL;
	bFlashScale       	      		: BOOL;
	bFlashScale4       		  		: BOOL;
	bFlashScale5        	  		: BOOL;
	bFlashingFreq2			  		: BOOL;
	bFlashScaleFast       	  		: BOOL;
	
//Master Control
	stMachineStatus					: ST_MachineStatusStruct;	
	stMasterControl					: ST_MasterControlStruct;
  	stStationSruct                  : ARRAY[0..1] OF ST_StandardStationStruct; (* Station 0 - Master
                                                                                  Station 1 - Leak test                                                           
                                                                                   *)

	
																				   
	stNest							: ST_Nest;                                                                        
	stAlarms                        : ARRAY [0..1] OF ST_Events;
	
	bManualModeTrigger				: BOOL;
	bFirstScan				:   BOOL;
	tFirstScan				:   TON;



	
																				   

END_VAR

// ---- GVLs/GVL_PERSIST.TcGVL
{attribute 'qualified_only'}
VAR_GLOBAL PERSISTENT
	
stPartsInspection			: ST_PartsInspection;
stUserLogHMI				: ARRAY[0..250] OF ST_UserLogHMI;
UserId						: UINT;
ast_i28LasResult            : ARRAY [0..250] OF st_i28LasResult;
nLeakTestID					: UINT;

nCycleNumber				: INT;
	
END_VAR

// ---- POUs/MAIN.TcPOU
PROGRAM MAIN
VAR
END_VAR

Main_Master();

END_PROGRAM

// ---- POUs/A_Master/Main_Master.TcPOU
PROGRAM Main_Master
VAR
	i                       :INT; //Int to handle user log index	
	k						:INT; //Int to handle user log index
	j						:INT;
	l						:INT;
	
	//////UserLog
	
	sUserGroupID			:	STRING;
	nSize					:	UDINT					:=9;
	nLen					:	UDINT					:=18;
	npos					:	UDINT					:=1;
	tonUserLogOut           :	Tc2_Standard.TON;
	fbStringFormatter       :	Tc2_Utilities.FB_FormatString;
	fbEventLogger			:	FB_EventLog;
	rUserLoggedIn			: 	R_TRIG;
	tUserLoggedIn			: 	TON;
	bFirstScan				:   BOOL;
	tFirstScan				:   TON;

	bUserLoggedIn			: 	BOOL;
	

	
	
	/////ShutDown&Quit
	closeChrome 			: 	NT_StartProcess;	
	ntShutdown					: TC2_Utilities.NT_Shutdown;
	ntError						: BOOL;
	ntBusy						: BOOL;
	ntErrorID					: UDINT;

	
	
	/////General

END_VAR

PRG_FaultHandling(aAlarms := GVL_Master.stAlarms );
PRG_Fault_LeakTest(aAlarms := GVL_Master.stAlarms);


PRG_MachineStatus();
PRG_MasterCycle(stStationStruct:= GVL_Master.stStationSruct[0]);
PRG_MasterSystemTime();
ACT_ShutdownAndQuit();
ACT_UserLog();
MapUnitEventsToHmi();
PRG_HMI();
PRG_Puls();
ACT_FirstScan();
PRG_TerminBoxInfo();

//gfggf




PRG_LeakTestEvents_Info();





//Stations
PRG_LeakTest(stStationStruct:= GVL_Master.stStationSruct[1]);




fbEventLogger(	bEnable       	:= PRG_MasterSystemTime.bReadyToRead AND GVL_MASTER.stMasterControl.bPowerUpTimerComplete,
			    sDateTime     	:= PRG_MasterSystemTime.sDateTimeSpaces,
			    aEventFlags   	:= GVL_HMI_GLOBAL.aEventFlags,
			    aEventTexts   	:= GVL_HMI_GLOBAL.aEventTexts,
			    aActiveEvents 	:= GVL_HMI_GLOBAL.aActiveEvents,
			    aEventLog     	:= GVL_HMI_GLOBAL.aEventLog,
				siDate			:= GVL_HMI_GLOBAL.sSystemDate,
				siTime			:= GVL_HMI_GLOBAL.sSystemTime,
				soDate			:= GVL_HMI_GLOBAL.aDateLog,
				soTime			:= GVL_HMI_GLOBAL.aTimeLog
);



 

IF GVL_MASTER.bFlashScale THEN
FOR j := 0 TO 39 DO
	
GVL_HMI_GLOBAL.stActiveEventsHMI[j].sActiveEvents := GVL_HMI_GLOBAL.aActiveEvents[j];
END_FOR
FOR l:=0 TO 250 DO
	
	GVL_HMI_GLOBAL.stAlarmHistory[l].sEventlog 	:= GVL_HMI_GLOBAL.aEventLog[l];
	GVL_HMI_GLOBAL.stAlarmHistory[l].sDate		:= GVL_HMI_GLOBAL.aDateLog[l];
	GVL_HMI_GLOBAL.stAlarmHistory[l].sTime		:= GVL_HMI_GLOBAL.aTimeLog[l];
END_FOR
ELSE 
	
j:=0; 
l:=0;

END_IF

ACTION ACT_FirstScan:
tFirstScan(IN := NOT bFirstScan, PT := T#5S);
END_ACTION

ACTION ACT_ShutdownAndQuit:
closeChrome(
    NetId := '',
    PathStr := 'C:\Windows\System32\mshta vbscript:Execute("CreateObject(""WScript.Shell"").Run ""powershell -c',
    DirName := 'C:\Windows\System32\WindowsPowerShell\v1.0',
    ComndLine := 'taskkill /F /IM chrome.exe /T"", 0: window.close")',
    Start := GVL_HMI_GLOBAL.bQuitHmi,
    TmOut := DEFAULT_ADS_TIMEOUT
);
 
GVL_HMI_GLOBAL.bQuitHmi:= FALSE;

ntShutdown(NETID := GVL_HMI_GLOBAL.ntAMSNetID, DELAY := 5, START := GVL_HMI_GLOBAL.bShutDown, BUSY => ntBusy, ERR => ntError, ERRID => ntErrorID);
END_ACTION

ACTION ACT_UserLog:

//Getting user group

Tc2_Utilities.DELETE2( ADR(GVL_HMI_GLOBAL.sUserGroup), ADR(sUserGroupID), NSize, Nlen, nPos) ;

IF sUserGroupID = 'Administ' THEN
	
	GVL_HMI_GLOBAL.sUserGroup2 := 'Administrator';

ELSE GVL_HMI_GLOBAL.sUserGroup2 := sUserGroupID;
	

END_IF


//Logout 

tonUserLogOut( IN := (sUserGroupID = 'Administ' OR sUserGroupID ='Engineer') AND GVL_HMI_GLOBAL.bUserLogedIntSignal , PT := T#10M);

IF tonUserLogOut.Q AND (sUserGroupID = 'Administ' OR sUserGroupID ='Engineer') THEN
	
	GVL_HMI_GLOBAL.bLogOut 	:= TRUE;

	ELSE GVL_HMI_GLOBAL.bLogOut := FALSE;

END_IF

tUserLoggedIn( IN := GVL_HMI_GLOBAL.bUserLogedIntSignal, PT := T#2S);

rUserLoggedIn( CLK := tUserLoggedIn.Q);


IF rUserLoggedIn.Q THEN
	
	FOR i :=200 TO 1 BY (-1) DO
		GVL_PERSIST.stUserLogHMI[i]	:= GVL_PERSIST.stUserLogHMI[i-1];
	END_FOR
	
	GVL_PERSIST.stUserLogHMI[0].UserLog := GVL_HMI_GLOBAL.sUserName;
	GVL_PERSIST.stUserLogHMI[0].UserLogTime := GVL_HMI_GLOBAL.sSystemTime;
	GVL_PERSIST.stUserLogHMI[0].UserLogDate := GVL_HMI_GLOBAL.sSystemDate;

END_IF
END_ACTION

METHOD MapUnitEventsToHMI : BOOL
VAR_INPUT
END_VAR

VAR
	i		:INT; 	//Unit index
	j		:INT;	//Unit event index
	k		:INT; 	//HMI event index	
END_VAR
//Set event texts first
IF GVL_Master.stAlarms[0].bEventTextsSet AND
   GVL_Master.stAlarms[1].bEventTextsSet AND
   NOT GVL_HMI_GLOBAL.bEventTextsSet 
THEN
	SetEventTexts();
		
	GVL_HMI_GLOBAL.bEventTextsSet := TRUE;
END_IF

//Map events from master and stations into HMI events
IF GVL_HMI_GLOBAL.bEventTextsSet THEN
	k := 0; 
	FOR i := 0 TO 4 DO
		FOR j := 0 TO 128 - 1 DO
			GVL_HMI_GLOBAL.aEventFlags[k] := GVL_Master.stAlarms[i].aEventFlags[j];
			k := k + 1;
		END_FOR
	END_FOR
END_IF
END_METHOD

METHOD SetEventTexts : BOOL
VAR_INPUT
END_VAR
VAR
	i				:INT; 	//Unit index
	j				:INT;	//HMI event index
	k				:INT;	//
END_VAR
//Set global event texts based on unit event texts (master and stations
k := 0;
FOR i := 0 TO 1 DO
	//For each unit (master, station1, station2)
	//Alarm texts
	FOR j := 0 TO 99 DO
		fbStringFormatter(	sFormat := 'Alarm No. %d - %s', 
					 	arg1 := F_INT(k), 
						arg2 := F_String(GVL_Master.stAlarms[i].aEventTexts[j]),
						sOut => GVL_HMI_GLOBAL.aEventTexts[k]);
						
		k := k + 1; //Increment global events index
	END_FOR
	
	//Messages
	FOR j := 100 TO 127 DO
		fbStringFormatter(	sFormat := 'Message No. %d - %s', 
					 		arg1 := F_INT(k), 
							arg2 := F_String(GVL_Master.stAlarms[i].aEventTexts[j]),
							sOut => GVL_HMI_GLOBAL.aEventTexts[k]);
							
		k := k + 1; //Increment global events index
	END_FOR
END_FOR
END_METHOD

END_PROGRAM

// ---- POUs/A_Master/PRG_FaultHandling.TcPOU
PROGRAM PRG_FaultHandling
VAR
	
	i							: INT;
	bFlagResetOn				: BOOL;
	bStationCycleFaultFlag		: BOOL;




END_VAR
VAR_IN_OUT

  aAlarms  : ARRAY[0..1] OF ST_Events;
END_VAR

ACT_FaultTrig();

(************************************** Faults reset **********************************************)
IF   GVL_HMI_GLOBAL.bResetButton THEN 
	FOR i := 0 TO 127 DO
		GVL_MASTER.stAlarms[0].aEventFlags[i] := FALSE;
	END_FOR
END_IF


//===============================================================
//Initialize event texts on first scan
IF NOT GVL_MASTER.stAlarms[0].bEventTextsSet THEN
	SetEventTexts();
	GVL_MASTER.stAlarms[0].bEventTextsSet := TRUE;
END_IF
IF NOT GVL_MASTER.stAlarms[0].bEventTextsSet THEN
	GVL_MASTER.stAlarms[0].bEventTextsSet := FALSE;
END_IF


(***************************************************************************************************)
//Immediate fault
GVL_MASTER.stAlarms[0].bImmediateFault := FALSE;
FOR i := 0 TO 32DO
	GVL_MASTER.stAlarms[0].bImmediateFault := GVL_MASTER.stAlarms[0].bImmediateFault OR GVL_MASTER.stAlarms[0].aEventFlags[i];
END_FOR

//Cycle stop fault
GVL_MASTER.stAlarms[0].bCycleStopFault := FALSE;
FOR i := 33 TO 79 DO
	GVL_MASTER.stAlarms[0].bCycleStopFault := GVL_MASTER.stAlarms[0].bCycleStopFault OR GVL_MASTER.stAlarms[0].aEventFlags[i];
END_FOR

//Cycle stop request
GVL_MASTER.stAlarms[0].bCycleStopRequest := FALSE;
FOR i := 80 TO 99 DO
	GVL_MASTER.stAlarms[0].bCycleStopRequest := GVL_MASTER.stAlarms[0].bCycleStopRequest OR GVL_MASTER.stAlarms[0].aEventFlags[i];
END_FOR


(**************************** Master Fault Monitors ***********************************************)
(* Station Immediate Fault Monitor *)
GVL_MASTER.stMasterControl.bNoStationImmediateFault := 	NOT GVL_MASTER.stAlarms[0].bImmediateFault AND NOT GVL_MASTER.stAlarms[1].bImmediateFault;

(**************************************************************************************************)
(**************************** Cycle stop falt  **************************************)
bStationCycleFaultFlag := NOT GVL_MASTER.stAlarms[0].bCycleStopFault AND NOT GVL_MASTER.stAlarms[1].bCycleStopFault;

(**************************** Master Immediate Fault Monitor **************************************)
GVL_MASTER.stMasterControl.bNoMachineImmediateFault := NOT GVL_MASTER.stAlarms[0].bImmediateFault AND NOT GVL_MASTER.stAlarms[1].bImmediateFault;

									
(**************************************************************************************************)

(* Master Cycle Stop Fault Monitor *)
GVL_MASTER.stMasterControl.bNoCycleStopFault := NOT GVL_MASTER.stAlarms[0].bCycleStopFault;

ACTION ACT_FaultTrig:
(**************************************************************************************************)
(**************************** Master Immediate Fault Stop *****************************************)
(**************************************************************************************************)

//Beckhoff EL1809 Not Operational
IF NOT GVL_MASTER.stMachineStatus.bSystemPowerUp AND GVL_IO.dwTerminalInfo[3].nTerminal_State<>8 THEN
	GVL_MASTER.stAlarms[0].aEventFlags[33] := TRUE;
END_IF
//Beckhoff EL2809 Not Operational
IF NOT GVL_MASTER.stMachineStatus.bSystemPowerUp AND GVL_IO.dwTerminalInfo[4].nTerminal_State<>8 THEN
	GVL_MASTER.stAlarms[0].aEventFlags[34] := TRUE;
END_IF

//System stopping timeout
GVL_MASTER.stAlarms[0].aEventTimers[38](IN := ( GVL_MASTER.stMachineStatus.bSystemStopping ), PT := T#20S);
IF GVL_MASTER.stAlarms[0].aEventTimers[38].Q THEN
	GVL_MASTER.stAlarms[0].aEventFlags[38] := TRUE;	
END_IF
//User not Log In
GVL_MASTER.stAlarms[0].aEventTimers[39](IN := (GVL_HMI_GLOBAL.sUserName=''), PT := T#40MS);
IF GVL_MASTER.stAlarms[0].aEventTimers[39].Q THEN
	GVL_MASTER.stAlarms[0].aEventFlags[39] := TRUE;	
END_IF
//User LOG-Off Timeout Manual Mode
GVL_MASTER.stAlarms[0].aEventTimers[40](IN:= ((GVL_HMI_GLOBAL.sUserName='') AND GVL_MASTER.stMachineStatus.bManualMode),PT:= T#1S); 
IF GVL_MASTER.stAlarms[0].aEventTimers[40].Q THEN
	GVL_MASTER.stAlarms[0].aEventFlags[40] := TRUE;
END_IF

//10 Min Auto cycle stop
IF PRG_MasterCycle.bAutoCycleStop  THEN //
	GVL_MASTER.stAlarms[0].aEventFlags[80] := TRUE;
END_IF
//Autocyle Timeout 
GVL_MASTER.stAlarms[0].aEventTimers[42](IN:= GVL_MASTER.stStationSruct[0].bStationInProgress, PT :=T#10M ); 
IF GVL_MASTER.stAlarms[0].aEventTimers[42].Q THEN
	GVL_MASTER.stAlarms[0].aEventFlags[42] := TRUE;
END_IF
//Clamp toggled before requested
IF GVL_MASTER.stStationSruct[0].nState > 1130 AND GVL_MASTER.stStationSruct[0].nState < 1700  //GVL_MASTER.stStationSruct[0].nState < 1900  **LAA 10092025 
	AND NOT GVL_IO.dw_T02_EL1809.iCalmpClosed THEN
	GVL_MASTER.stAlarms[0].aEventFlags[43] := TRUE;
END_IF
//Nest taken before requested
IF GVL_MASTER.stStationSruct[0].nState > 1000 AND GVL_MASTER.stStationSruct[0].nState < 1900 
	AND NOT GVL_IO.dw_T02_EL1809.iPartPresent AND GVL_IO.dw_T02_EL1809.iCalmpClosed  THEN  //**LA 04092025
	GVL_MASTER.stAlarms[0].aEventFlags[44] := TRUE;
END_IF
//Press Acknowledge
IF GVL_HMI_GLOBAL.bAutoCycleFaultDialog THEN
	GVL_MASTER.stAlarms[0].aEventFlags[45] := TRUE;
END_IF


//Remove Nest   //**LA 12092025
IF GVL_HMI_GLOBAL.bStartButton AND NOT PRG_Mastercycle.biClamp AND PRG_Mastercycle.biPartPresent THEN 
	GVL_MASTER.stAlarms[0].aEventFlags[100] := TRUE;
	ELSIF NOT PRG_Mastercycle.biPartPresent THEN 
		GVL_MASTER.stAlarms[0].aEventFlags[100] := FALSE;
END_IF

//Release Clamp //**LA 12092025
IF GVL_HMI_GLOBAL.bStartButton AND PRG_Mastercycle.biClamp AND NOT PRG_Mastercycle.biPartPresent AND GVL_MASTER.stMachineStatus.bSystemReadyToStart THEN 
	GVL_MASTER.stAlarms[0].aEventFlags[101] := TRUE;
	ELSIF NOT PRG_Mastercycle.biClamp THEN 
		GVL_MASTER.stAlarms[0].aEventFlags[101] := FALSE;
END_IF

//Releas Clamp and Remove Nest //**LA 12092025
IF GVL_HMI_GLOBAL.bStartButton AND PRG_Mastercycle.biClamp AND PRG_Mastercycle.biPartPresent AND GVL_MASTER.stMachineStatus.bSystemReadyToStart THEN
	GVL_MASTER.stAlarms[0].aEventFlags[102] := TRUE;
	ELSIF  NOT PRG_Mastercycle.biClamp AND NOT PRG_Mastercycle.biPartPresent THEN
		GVL_MASTER.stAlarms[0].aEventFlags[102] := FALSE;
END_IF
END_ACTION

METHOD PRIVATE SetEventTexts : BOOL
VAR_INPUT
END_VAR
//Immediate Faults
GVL_MASTER.stAlarms[0].aEventTexts[0] := 'SPARE';
GVL_MASTER.stAlarms[0].aEventTexts[1] := 'SPARE';
GVL_MASTER.stAlarms[0].aEventTexts[2] := 'SPARE';
GVL_MASTER.stAlarms[0].aEventTexts[3] := 'SPARE';
GVL_MASTER.stAlarms[0].aEventTexts[4] := '';
GVL_MASTER.stAlarms[0].aEventTexts[5] := '';
GVL_MASTER.stAlarms[0].aEventTexts[6] := '';
GVL_MASTER.stAlarms[0].aEventTexts[7] := '';
GVL_MASTER.stAlarms[0].aEventTexts[8] := '';
GVL_MASTER.stAlarms[0].aEventTexts[9] := '';
GVL_MASTER.stAlarms[0].aEventTexts[10] := '';
GVL_MASTER.stAlarms[0].aEventTexts[10] := ''; 
GVL_MASTER.stAlarms[0].aEventTexts[11] := '';
GVL_MASTER.stAlarms[0].aEventTexts[12] := '';
GVL_MASTER.stAlarms[0].aEventTexts[13] := '';
GVL_MASTER.stAlarms[0].aEventTexts[14] := '';
GVL_MASTER.stAlarms[0].aEventTexts[15] := '';


//Cycle stop fault

GVL_MASTER.stAlarms[0].aEventTexts[33] := 'Beckhoff EL1809 Not Operational';
GVL_MASTER.stAlarms[0].aEventTexts[34] := 'Beckhoff EL2809 Not Operational';
GVL_MASTER.stAlarms[0].aEventTexts[35] := '';
GVL_MASTER.stAlarms[0].aEventTexts[36] := '';
GVL_MASTER.stAlarms[0].aEventTexts[37] := '';
GVL_MASTER.stAlarms[0].aEventTexts[38] := 'Master - Stopping timeout';
GVL_MASTER.stAlarms[0].aEventTexts[39] := 'User Not Log IN';
GVL_MASTER.stAlarms[0].aEventTexts[40] := 'User Log-Off Timeout Manual Mode'; 
GVL_MASTER.stAlarms[0].aEventTexts[41] := '';
GVL_MASTER.stAlarms[0].aEventTexts[42] := 'Autocyle Timeout' ;
GVL_MASTER.stAlarms[0].aEventTexts[43] := 'Clamp toggled before requested';
GVL_MASTER.stAlarms[0].aEventTexts[44] := 'Nest taken before requested';
GVL_MASTER.stAlarms[0].aEventTexts[45] := 'Press Acknowledge';
GVL_MASTER.stAlarms[0].aEventTexts[46] := '';
GVL_MASTER.stAlarms[0].aEventTexts[47] := '';
GVL_MASTER.stAlarms[0].aEventTexts[48] := '';
GVL_MASTER.stAlarms[0].aEventTexts[59] := '';
GVL_MASTER.stAlarms[0].aEventTexts[50] := '';

//Cycle Stop Requests

GVL_MASTER.stAlarms[0].aEventTexts[80] := 'Machine Cycle Stop 10 Min Not Use Timeout';
GVL_MASTER.stAlarms[0].aEventTexts[81] := '';
GVL_MASTER.stAlarms[0].aEventTexts[82] := '';

GVL_MASTER.stAlarms[0].aEventTexts[84] := '';
GVL_MASTER.stAlarms[0].aEventTexts[85] := '';
GVL_MASTER.stAlarms[0].aEventTexts[86] := '';
GVL_MASTER.stAlarms[0].aEventTexts[87] := ''; 
GVL_MASTER.stAlarms[0].aEventTexts[88] := '';
GVL_MASTER.stAlarms[0].aEventTexts[89] := '';

// Message  //**LA 12092025
GVL_MASTER.stAlarms[0].aEventTexts[100] := 'Remove Nest';
GVL_MASTER.stAlarms[0].aEventTexts[101] := 'Release Clamp';
GVL_MASTER.stAlarms[0].aEventTexts[102] := 'Release Clamp and Remove Nest';
END_METHOD

END_PROGRAM

// ---- POUs/A_Master/PRG_MasterCycle.TcPOU
PROGRAM PRG_MasterCycle
VAR
	
		tonCaseTimDelay    	: ARRAY [1..20] OF Tc2_Standard.TON;
	    rtrigCaseTriger    	: ARRAY [1..10] OF Tc2_Standard.R_TRIG;
		ftrigCaseTriger		: ARRAY [1..10] OF Tc2_Standard.F_TRIG;
	   	rtrigFaultMachine  	: Tc2_Standard.R_TRIG;	
		
		biClamp				: BOOL;
		biPartPresent		: BOOL;
		


		bAutoCycleStop		: BOOL;
		
		bCycleFlag			: BOOL;
		bGreenLED			: BOOL;
		bRedLED				: BOOL;
		bEndCycleFlag		: BOOL;
		bStationsStopped	: BOOL;
		bLeakTestCompleteFlag : BOOL;
		i					: DINT;
		
		


END_VAR
VAR_IN_OUT
	stStationStruct          : ST_StandardStationStruct;
END_VAR

ACT_LinkIO();
ACT_TimTrig();
stStationStruct.bStationInProgress := stStationStruct.nState>=1100 AND stStationStruct.nState<=1700;

IF stStationStruct.nState <700 OR (stStationStruct.nState > 1700 AND stStationStruct.nState <4000) OR stStationStruct.nState > 4000 THEN
	GVL_HMI_GLOBAL.sActualProcess := ""; 
	GVL_MASTER.stNest.bPiecePass 	:= FALSE;
	GVL_MASTER.stNest.bPieceReject 	:= FALSE;
	bGreenLED						:= FALSE;
	bRedLED							:= FALSE;
END_IF

IF rtrigCaseTriger[3].Q THEN
GVL_PERSIST.stPartsInspection.nPartsGood:= GVL_PERSIST.stPartsInspection.nPartsGood +1;
GVL_PERSIST.stPartsInspection.nTotalPartsGood := GVL_PERSIST.stPartsInspection.nTotalPartsGood+1;
ELSIF GVL_HMI_GLOBAL.bResetGoodParts THEN
GVL_PERSIST.stPartsInspection.nPartsGood:=0;	
END_IF


IF rtrigCaseTriger[4].Q THEN
	GVL_PERSIST.stPartsInspection.nPartsFailed:=GVL_PERSIST.stPartsInspection.nPartsFailed+1;
	GVL_PERSIST.stPartsInspection.nTotalPartsFailed:= GVL_PERSIST.stPartsInspection.nTotalPartsFailed+1;
ELSIF GVL_HMI_GLOBAL.bResetFailedParts THEN
	GVL_PERSIST.stPartsInspection.nPartsFailed:=0;
END_IF

IF stStationStruct.nState < 700 THEN
	 GVL_HMI_GLOBAL.sMessageToOperator := "Press Reset Button to Home Machine";
END_IF

CASE stStationStruct.nState OF
	
100: 
   bAutoCycleStop := FALSE;
IF NOT GVL_MASTER.stMachineStatus.bSystemPowerUp THEN
	stStationStruct.nState := 200;
END_IF
200:
IF GVL_MASTER.stMachineStatus.bSystemInitialising THEN
	stStationStruct.nState := 300;
END_IF
300:
   GVL_Master.stStationSruct[1].bStationInitRequest := TRUE;
   
IF GVL_Master.stStationSruct[1].bStationInitRequest THEN
	stStationStruct.nState := 400;
END_IF
400:
IF NOT GVL_Master.stStationSruct[1].bStationInitRequest THEN
	stStationStruct.nState := 500;   
END_IF 
500:
   GVL_Master.stStationSruct[1].bStationAcknowledge := TRUE;
IF   GVL_Master.stStationSruct[1].bStationAcknowledge THEN
     stStationStruct.nState := 600;
END_IF
600:
IF GVL_Master.stStationSruct[1].bStationHomed THEN
   GVL_Master.stStationSruct[1].bStationAcknowledge := FALSE;

   stStationStruct.nState := 700;
END_IF
700: // All Station Homed and waiting for Autocycle 
   bAutoCycleStop := FALSE;
   GVL_HMI_GLOBAL.sActualProcess := "Waiting for Autocycle";
   GVL_HMI_GLOBAL.sMessageToOperator := "Press Start Button to Autocycle";
IF GVL_Master.stMachineStatus.bSystemAutoCycle THEN
	stStationStruct.nState := 800;
ELSIF GVL_Master.stMachineStatus.bManualMode THEN
      stStationStruct.nState := 4000;
ELSIF GVL_Master.stMachineStatus.bSystemStopping AND NOT bStationsStopped  THEN
      stStationStruct.nState := 5000;
ELSIF GVL_Master.stMachineStatus.bCycleStopFault OR GVL_Master.stMachineStatus.bImmediateFault THEN
      stStationStruct.nState := 6000;	  
END_IF

IF tonCaseTimDelay[9].Q THEN
	stStationStruct.nState := 1000;
END_IF
800:
stStationStruct.nState := 1000;
1000: // System Autocycle

IF biPartPresent THEN
	GVL_HMI_GLOBAL.sMessageToOperator := "Remove Nest";
ELSE GVL_HMI_GLOBAL.sMessageToOperator := "Insert Nest";
END_IF


IF  rtrigCaseTriger [5].Q  AND NOT bEndCycleFlag THEN
	GVL_MASTER.stNest.bPiecePass 	:= FALSE;
	GVL_MASTER.stNest.bPieceReject 	:= FALSE;
	GVL_MASTER.stNest.bNestPartProced := FALSE;
	GVL_MASTER.stNest.sLeakHMI 		:= "";
	GVL_MASTER.stNest.sPieceHMI 	:= "";
	bCycleFlag						:= TRUE;
	GVL_HMI_GLOBAL.bResetPassAndFail:= TRUE;
	GVL_HMI_GLOBAL.sActualProcess := "";
	bGreenLED						:= FALSE;
	bRedLED							:= FALSE;
	GVL_HMI_GLOBAL.bRejectPieceAcknowledge := FALSE;
	stStationStruct.nState 			:= 1110;
ELSIF GVL_Master.stMachineStatus.bSystemStopping  THEN
      stStationStruct.nState := 5000;
ELSIF tonCaseTimDelay[10].Q THEN
	  bAutoCycleStop := TRUE;
      stStationStruct.nState := 5000;	
END_IF
1110:
IF GVL_HMI_GLOBAL.bStopperPressEnable THEN
	GVL_HMI_GLOBAL.sMessageToOperator := "Toggle clamp to Press Stopper";
ELSE
	GVL_HMI_GLOBAL.sMessageToOperator := "Toggle clamp to Start Leak Test";
END_IF

IF rtrigCaseTriger [1].Q AND NOT GVL_HMI_GLOBAL.bStopperPressEnable THEN
	stStationStruct.nState 			:= 1130;
ELSIF rtrigCaseTriger [1].Q AND GVL_HMI_GLOBAL.bStopperPressEnable THEN
	stStationStruct.nState 			:= 1120;
ELSIF GVL_Master.stMachineStatus.bSystemStopping  THEN
      stStationStruct.nState := 5000;
ELSIF tonCaseTimDelay[10].Q THEN
	  bAutoCycleStop := TRUE;
      stStationStruct.nState := 5000;	
ELSIF rtrigCaseTriger [6].Q THEN 			 // **LA 04092025
	stStationStruct.nState 			:= 1000; // **LA 04092025
END_IF
1120:
//GVL_HMI_GLOBAL.sMessageToOperator := "Toggle clamp to begin process";
//IF rtrigCaseTriger [1].Q THEN
//	stStationStruct.nState 			:= 1130;
//END_IF
	GVL_HMI_GLOBAL.sMessageToOperator := "Release clamp";
IF rtrigCaseTriger [7].Q THEN
	stStationStruct.nState 			:= 1125;
END_IF
1125: 
GVL_HMI_GLOBAL.sMessageToOperator := "Relocate part and toggle clamp to Start Leak Test";
	IF rtrigCaseTriger [1].Q THEN
	stStationStruct.nState 			:= 1130;
END_IF

1130:
GVL_HMI_GLOBAL.sMessageToOperator := "Process in progress";
IF tonCaseTimDelay[13].Q THEN
	GVL_HMI_GLOBAL.bResetPassAndFail:= FALSE;
	stStationStruct.nState 			:= 1142;
END_IF

//Leak test
1142: 
	GVL_HMI_GLOBAL.sMessageToOperator := "Process in progress";
	GVL_HMI_GLOBAL.sActualProcess := "Leak test process"; 
	GVL_Master.stStationSruct[1].bStationRequest := TRUE;
	stStationStruct.nState := 1144;
1144:
IF GVL_Master.stStationSruct[1].bStationInProgress THEN
	stStationStruct.nState := 1146;
END_IF
1146:
IF GVL_Master.stStationSruct[1].bStationComplete THEN
	bLeakTestCompleteFlag := TRUE;
END_IF

IF  bLeakTestCompleteFlag AND NOT GVL_Master.stMachineStatus.bSystemStopping THEN
	stStationStruct.nState := 1152;
ELSIF GVL_Master.stMachineStatus.bSystemStopping THEN
	stStationStruct.nState := 5000;
END_IF

1152: 
	GVL_MASTER.stNest.bNestPartProced 	:= TRUE;
	bLeakTestCompleteFlag				:= FALSE;
IF tonCaseTimDelay[12].Q THEN
	stStationStruct.nState := 1220;
END_IF
	
1220:
IF  GVL_MASTER.stNest.bLeakPass THEN
	GVL_MASTER.stNest.bPiecePass 	:= TRUE;
	GVL_MASTER.stNest.bPieceReject 	:= FALSE;
	GVL_MASTER.stNest.sPieceHMI 	:= "Pass";
	bGreenLED						:= TRUE;
	bRedLED							:= FALSE;
ELSE 
	GVL_MASTER.stNest.sPieceHMI 	:= "Fail";
	GVL_MASTER.stNest.bPiecePass 	:= FALSE;
	GVL_MASTER.stNest.bPieceReject 	:= TRUE;
	bGreenLED						:= FALSE;
	bRedLED							:= TRUE;
END_IF
GVL_MASTER.stNest.sDate := GVL_HMI_GLOBAL.sSystemDate;
GVL_MASTER.stNest.sTime := GVL_HMI_GLOBAL.sSystemTime;

IF rtrigCaseTriger [8].Q THEN	
	
	FOR i :=200 TO 2 BY (-1) DO
		GVL_HMI_GLOBAL.aStatistics[i]	:= GVL_HMI_GLOBAL.aStatistics[i-1];
	END_FOR
	
	GVL_HMI_GLOBAL.aStatistics[1] := GVL_MASTER.stNest;
END_IF

IF tonCaseTimDelay[11].Q THEN
	stStationStruct.nState := 1500;
END_IF

1500:
IF GVL_Master.stStationSruct[1].bStationNotMoving  THEN
	stStationStruct.nState := 1550;
END_IF
1550:
IF  GVL_MASTER.stNest.bPiecePass THEN	
	stStationStruct.nState := 1600;
ELSIF  GVL_MASTER.stNest.bPieceReject AND GVL_HMI_GLOBAL.bRejectPieceAcknowledge THEN
	stStationStruct.nState := 1600;
END_IF

1600:
bEndCycleFlag	:= TRUE;
GVL_HMI_GLOBAL.sMessageToOperator := "Cycle Complete";
IF NOT GVL_MASTER.stMachineStatus.bSystemStopping  THEN 
	stStationStruct.nState := 1700;
	//stStationStruct.nState := 1000;
ELSE 
    stStationStruct.nState := 5000;	
END_IF

1700: 
GVL_HMI_GLOBAL.sMessageToOperator := "Release clamp"; 
IF rtrigCaseTriger [7].Q THEN 
	stStationStruct.nState := 1000;
END_IF
4000: 
IF NOT GVL_MASTER.stMachineStatus.bManualMode THEN
	stStationStruct.nState := 700;	
ELSIF GVL_MASTER.stMachineStatus.bCycleStopFault OR GVL_MASTER.stMachineStatus.bImmediateFault THEN
      stStationStruct.nState := 6000;		
END_IF

//stopping
5000:
	GVL_Master.stStationSruct[1].bNoCycleStopRequest := FALSE;
	
IF tonCaseTimDelay[6].Q AND (GVL_Master.stStationSruct[1].nState = 1000) THEN
	bAutoCycleStop := FALSE;	
	stStationStruct.nState := 700;

	
END_IF

6000:
IF tonCaseTimDelay[1].Q THEN
	GVL_Master.stStationSruct[1].bStationInitRequest := FALSE;
	GVL_Master.stStationSruct[1].bStationRequest := FALSE;
	GVL_Master.stStationSruct[1].bStationAbort := TRUE;
	stStationStruct.nState := 100;
END_IF


END_CASE

//++++++++++++++++++++++++++++++++++++++++++++++++++++++++++++++++++++++++++++++++++++++++++++++++++++++++++++++++++++++++++++++++++++++

IF rtrigFaultMachine.Q THEN
   stStationStruct.nState := 6000;	  
END_IF

IF  (stStationStruct.nState = 4000) OR (stStationStruct.nState = 5000) OR (stStationStruct.nState = 6000) THEN
   GVL_Master.stStationSruct[1].bStationAcknowledge := FALSE;
   GVL_Master.stStationSruct[1].bStationInitRequest := FALSE;
END_IF

ACTION ACT_LinkIO:
// Initialisation Progres
IF GVL_Master.stStationSruct[1].bStationInProgressInit THEN
	GVL_Master.stStationSruct[1].bStationInitRequest := FALSE;
END_IF
// Cycle Progres
IF GVL_Master.stStationSruct[1].bStationInProgress THEN
	GVL_Master.stStationSruct[1].bStationRequest := FALSE;
END_IF

// Abort Station
IF GVL_Master.stStationSruct[1].nState = 100 THEN
	GVL_Master.stStationSruct[1].bStationAbort := FALSE;
END_IF

IF (GVL_Master.stStationSruct[1].nState = 100) OR (GVL_Master.stStationSruct[1].nState = 1000) THEN
	GVL_Master.stStationSruct[1].bNoCycleStopRequest := TRUE;
END_IF


IF  (GVL_Master.stStationSruct[1].nState = 700)  THEN
	bStationsStopped := TRUE;
ELSE bStationsStopped := FALSE;

END_IF

GVL_MASTER.stMasterControl.bAllStationsCycledStopped := (GVL_Master.stStationSruct[1].nState = 1000) AND  stStationStruct.nState=700;
										 
	biClamp									:= GVL_IO.dw_T02_EL1809.iCalmpClosed;
	biPartPresent							:=  GVL_IO.dw_T02_EL1809.iPartPresent;
	GVL_MASTER.stNest.bNestPresent			:= GVL_IO.dw_T02_EL1809.iCalmpClosed;
	GVL_IO.dw_T03_EL2809.qPassIndicatorGreen:= bGreenLED;
	GVL_IO.dw_T03_EL2809.qRejectIndicatorRed:= bRedLED;
	
IF ftrigCaseTriger[1].Q THEN
	bEndCycleFlag							:= FALSE;
END_IF
	

GVL_HMI_GLOBAL.nGeneralCycTime := (TIME_TO_DINT(GVL_MASTER.stAlarms[0].aEventTimers[42].ET))/1000;
END_ACTION

ACTION ACT_TimTrig:
tonCaseTimDelay[1](IN:= (stStationStruct.nState = 6000),PT:=T#100MS); //
tonCaseTimDelay[2](IN:= (stStationStruct.nState = 5000),PT:=T#100MS); //
tonCaseTimDelay[3](IN:= (stStationStruct.nState = 1100),PT:=T#40MS);  //
tonCaseTimDelay[4](IN:= (stStationStruct.nState = 1140),PT:=T#250MS);
tonCaseTimDelay[5](IN:= (stStationStruct.nState = 1900),PT:=T#250MS);
tonCaseTimDelay[6](IN:= (stStationStruct.nState = 5000),PT:=T#250MS);
tonCaseTimDelay[7](IN:= (stStationStruct.nState = 1340),PT:=T#200MS);
tonCaseTimDelay[8](IN:= (stStationStruct.nState = 1320),PT:=T#500MS);
tonCaseTimDelay[9](IN:= (stStationStruct.nState = 800),PT:=T#3S);
tonCaseTimDelay[10](IN:= (stStationStruct.nState = 1000),PT:=T#10M);
tonCaseTimDelay[11](IN:= (stStationStruct.nState = 1220),PT:=T#1S);
tonCaseTimDelay[12](IN:= stStationStruct.nState = 1152,PT:=T#1S );
tonCaseTimDelay[13](IN:=(stStationStruct.nState = 1130),PT:=T#1S );
tonCaseTimDelay[14](IN:=,PT:=T#1S);
tonCaseTimDelay[15](IN:= );
tonCaseTimDelay[16](IN:= );
tonCaseTimDelay[17](IN:= );
tonCaseTimDelay[18](IN:= );
tonCaseTimDelay[19](IN:= );
tonCaseTimDelay[20](IN:= );

rtrigCaseTriger [1](CLK:= biClamp);
rtrigCaseTriger [2](CLK:= tonCaseTimDelay[2].Q);
rtrigCaseTriger [3](CLK:= GVL_MASTER.stNest.bPiecePass);
rtrigCaseTriger [4](CLK:= GVL_MASTER.stNest.bPieceReject);
rtrigCaseTriger [5](CLK:= biPartPresent );
rtrigCaseTriger [6](CLK:= (stStationStruct.nState = 1110) AND NOT biPartPresent AND NOT biClamp );  //LA** 04092025
rtrigCaseTriger [7](CLK:= NOT biClamp);
rtrigCaseTriger [8](CLK:= (stStationStruct.nState = 1220));
rtrigCaseTriger [9](CLK:= );
rtrigCaseTriger [10](CLK:= );
rtrigFaultMachine(CLK:= GVL_MASTER.stMachineStatus.bCycleStopFault OR GVL_MASTER.stMachineStatus.bImmediateFault);

ftrigCaseTriger [1](CLK:= biPartPresent );
END_ACTION

END_PROGRAM

// ---- POUs/C_LeakTest/PRG_Fault_LeakTest.TcPOU
PROGRAM PRG_Fault_LeakTest
VAR
	


				i						: INT;
END_VAR
VAR_IN_OUT

  aAlarms  : ARRAY[0..1] OF ST_Events;
END_VAR

ACT_FaultTrig();

(************************************** Faults reset **********************************************)
IF   GVL_HMI_GLOBAL.bResetButton THEN 
	FOR i := 0 TO 127 DO
		GVL_MASTER.stAlarms[1].aEventFlags[i] := FALSE;
	END_FOR
END_IF
//===============================================================
//Initialize event texts on first scan
IF NOT GVL_MASTER.stAlarms[1].bEventTextsSet THEN
	SetEventTexts();
	GVL_MASTER.stAlarms[1].bEventTextsSet := TRUE;
END_IF


(***************************************************************************************************)
//Immediate fault
GVL_MASTER.stAlarms[1].bImmediateFault := FALSE;
FOR i := 0 TO 32DO
	GVL_MASTER.stAlarms[1].bImmediateFault := GVL_MASTER.stAlarms[1].bImmediateFault OR GVL_MASTER.stAlarms[1].aEventFlags[i];
END_FOR

//Cycle stop fault
GVL_MASTER.stAlarms[1].bCycleStopFault := FALSE;
FOR i := 33 TO 79 DO
	GVL_MASTER.stAlarms[1].bCycleStopFault := GVL_MASTER.stAlarms[1].bCycleStopFault OR GVL_MASTER.stAlarms[1].aEventFlags[i];
END_FOR
//Cycle stop Request
GVL_MASTER.stAlarms[1].bCycleStopRequest := FALSE;
FOR i := 80 TO 99 DO
	GVL_MASTER.stAlarms[1].bCycleStopRequest := GVL_MASTER.stAlarms[1].bCycleStopRequest OR GVL_MASTER.stAlarms[1].aEventFlags[i];
END_FOR

ACTION ACT_FaultTrig:
(**************************************************************************************************)
(**************************** Master Immediate Fault Stop *****************************************)
(**************************************************************************************************)
(* Copy Safety Immediate Stop Faults to Master Immediate Stop Faults *)
(* *)

//Leak Station Not Homed Timeout
GVL_MASTER.stAlarms[1].aEventTimers[0](IN:= (GVL_Master.stStationSruct[1].nState>=200 AND GVL_Master.stStationSruct[1].nState<=900) ,PT:=T#5S);																	
IF GVL_MASTER.stAlarms[1].aEventTimers[0].Q THEN //
	GVL_MASTER.stAlarms[1].aEventFlags[0] := TRUE;
END_IF
//Leak Station Cycle Timeout
GVL_MASTER.stAlarms[1].aEventTimers[1](IN:= (GVL_Master.stStationSruct[1].nState>=1100 AND GVL_Master.stStationSruct[1].nState<=1900) ,PT:=T#40S);
IF GVL_MASTER.stAlarms[1].aEventTimers[1].Q THEN // 
	GVL_MASTER.stAlarms[1].aEventFlags[1] := TRUE;
END_IF
//Leak Error
GVL_MASTER.stAlarms[1].aEventTimers[2](IN := (NOT PRG_LeakTest.bLeakTesterNoError),PT:=T#100MS);
IF GVL_MASTER.stAlarms[1].aEventTimers[2].Q THEN //
	GVL_MASTER.stAlarms[1].aEventFlags[2] := TRUE;
END_IF
END_ACTION

METHOD SetEventTexts : BOOL
VAR_INPUT
END_VAR
//Immediate Faults
GVL_MASTER.stAlarms[1].aEventTexts[0] := 'Leak Station Not Homed Timeout';
GVL_MASTER.stAlarms[1].aEventTexts[1] := 'Leak Station Cycle Timeout';
GVL_MASTER.stAlarms[1].aEventTexts[2] := 'Leak Error';
GVL_MASTER.stAlarms[1].aEventTexts[3] := 'More than 2 Consecutive rejects';
GVL_MASTER.stAlarms[1].aEventTexts[4] := '';
GVL_MASTER.stAlarms[1].aEventTexts[5] := '';
GVL_MASTER.stAlarms[1].aEventTexts[6] := '';
GVL_MASTER.stAlarms[1].aEventTexts[7] := '';
GVL_MASTER.stAlarms[1].aEventTexts[8] := '';
GVL_MASTER.stAlarms[1].aEventTexts[9] := ''; 
GVL_MASTER.stAlarms[1].aEventTexts[10] := ''; 
GVL_MASTER.stAlarms[1].aEventTexts[11] := '';
GVL_MASTER.stAlarms[1].aEventTexts[12] := '';
GVL_MASTER.stAlarms[1].aEventTexts[13] := '';
GVL_MASTER.stAlarms[1].aEventTexts[14] := '';
GVL_MASTER.stAlarms[1].aEventTexts[15] := '';
GVL_MASTER.stAlarms[1].aEventTexts[16] := '';
GVL_MASTER.stAlarms[1].aEventTexts[17] := '';
GVL_MASTER.stAlarms[1].aEventTexts[18] := '';
GVL_MASTER.stAlarms[1].aEventTexts[19] := '';
GVL_MASTER.stAlarms[1].aEventTexts[20] := '';
GVL_MASTER.stAlarms[1].aEventTexts[21] := '';
GVL_MASTER.stAlarms[1].aEventTexts[22] := '';
GVL_MASTER.stAlarms[1].aEventTexts[28] := '';
GVL_MASTER.stAlarms[1].aEventTexts[29] := '';
GVL_MASTER.stAlarms[1].aEventTexts[30] := '';

//Cycle Stop Requests

GVL_MASTER.stAlarms[1].aEventTexts[80] := '';
GVL_MASTER.stAlarms[1].aEventTexts[81] := '';
GVL_MASTER.stAlarms[1].aEventTexts[82] := '';

GVL_MASTER.stAlarms[1].aEventTexts[84] := '';
GVL_MASTER.stAlarms[1].aEventTexts[85] := '';
GVL_MASTER.stAlarms[1].aEventTexts[86] := '';
GVL_MASTER.stAlarms[1].aEventTexts[87] := ''; 
GVL_MASTER.stAlarms[1].aEventTexts[88] := '';
GVL_MASTER.stAlarms[1].aEventTexts[89] := '';

//Master Messages

GVL_MASTER.stAlarms[1].aEventTexts[100] := '';
GVL_MASTER.stAlarms[1].aEventTexts[101] := '';
GVL_MASTER.stAlarms[1].aEventTexts[102] := '';
GVL_MASTER.stAlarms[1].aEventTexts[103] := '';
GVL_MASTER.stAlarms[1].aEventTexts[104] := '';
GVL_MASTER.stAlarms[1].aEventTexts[105] := '';
GVL_MASTER.stAlarms[1].aEventTexts[106] := '';
END_METHOD

END_PROGRAM

// ---- POUs/C_LeakTest/PRG_LeakTest.TcPOU
PROGRAM PRG_LeakTest
VAR
		rPressure			: REAL; //**LA 10092025
		TonCaseDelay  		: ARRAY[1..10] OF Tc2_Standard.TON;
		rtrigCaseTriger  	: ARRAY [1..10] OF Tc2_Standard.R_TRIG;
		
		bLeakTesterNoError	: BOOL;
		uCurrentProgramID	: USINT;
		uSetProgramID		: USINT;
		bProgramAccepted	: BOOL;
		bProgramRejected	: BOOL;
		bInstrumentReady	: BOOL;
		bStart				: BOOL;
		bStop				: BOOL;
		bClearErrorIns		: BOOL;
		bTestActiveLiveData	: BOOL;
		nLiveMeasID			: UDINT;
		nLastMeasID			: UDINT;
		bJobPass			: BOOL;
		bJobFailed			: BOOL;
		nConsParts			: INT;






END_VAR
VAR_IN_OUT
	stStationStruct          : ST_StandardStationStruct;
END_VAR

ACT_IOLink();
ACT_TimTrig();

(************** Station in Home Position **************************)
stStationStruct.bStationHomed :=  (stStationStruct.nState = 1000);

(******************************************************************)
stStationStruct.bStationComplete := stStationStruct.nState = 1900;
stStationStruct.bStationHomingRequest := stStationStruct.nState = 200;
stStationStruct.bStationWaitOnRequest := stStationStruct.nState = 1000; 
stStationStruct.bStationInitDone := stStationStruct.nState = 900;
stStationStruct.bStationInProgressInit := stStationStruct.nState >= 200 AND stStationStruct.nState <= 900;
stStationStruct.bStationInProgress :=  stStationStruct.nState > 1000 AND stStationStruct.nState < 1900;
stStationStruct.bStationWaitOnInit := stStationStruct.nState = 100; 
//stStationStruct.bStationAcknowledge := stStationStruct.nState = 200 OR stStationStruct.nState = 1100;
stStationStruct.bStationNotMoving := stStationStruct.nState = 100 OR stStationStruct.nState = 1000 OR stStationStruct.nState = 1900;
(******************************************************************)

bClearErrorIns := GVL_HMI_GLOBAL.bResetButton;

(***************************************)

IF rtrigCaseTriger[3].Q THEN
	stStationStruct.nState := 100;
END_IF

(***************************************)


CASE stStationStruct.nState OF
100: 
IF stStationStruct.bStationInitRequest THEN
	 stStationStruct.nState := 120;
END_IF
120:
bClearErrorIns := TRUE;
IF bClearErrorIns THEN
	stStationStruct.nState := 160;
END_IF
160:
IF tonCaseDelay[2].Q THEN
	bClearErrorIns := FALSE;
	stStationStruct.nState := 180;
END_IF
180: // Check if error 
IF bLeakTesterNoError THEN
	 stStationStruct.nState := 400;
END_IF
400:
IF tonCaseDelay[1].Q THEN
	stStationStruct.nState := 800;
END_IF
800:
IF bInstrumentReady THEN
	stStationStruct.nState := 900;
END_IF
900:
IF stStationStruct.bStationAcknowledge THEN
	stStationStruct.nState := 1000;
END_IF

1000: // Waiting for request 
IF GVL_HMI_GLOBAL.bResetPassAndFail THEN
	GVL_MASTER.stNest.bLeakPass 	:= FALSE;
   GVL_MASTER.stNest.sLeakHMI 	:= "";
   GVL_MASTER.stNest.bLeakReject := FALSE;
END_IF

IF stStationStruct.bStationRequest AND stStationStruct.bNoCycleStopRequest THEN
   stStationStruct.nState := 1100;  
ELSIF (stStationStruct.bStationManualRequestHMI OR GVL_MASTER.bManualModeTrigger) AND stStationStruct.bNoCycleStopRequest THEN
   stStationStruct.nState := 4000; // Manual Mode
ELSIF stStationStruct.bStationAbort THEN
	   stStationStruct.nState := 100;	   
END_IF
1100: // Check Ready
bStart						:= FALSE;
GVL_MASTER.stNest.bLeakPass := FALSE;
GVL_MASTER.stNest.sLeakHMI 	:= "";
IF bInstrumentReady THEN
	stStationStruct.nState := 1140; 
ELSE
	stStationStruct.nState := 9000;
END_IF
1140://Check status of intrument
IF bLeakTesterNoError THEN
	stStationStruct.nState := 1200;
END_IF
1200: 
bStart := TRUE;
IF  tonCaseDelay[3].Q THEN
	stStationStruct.nState := 1220;
END_IF
1220:
bStart := FALSE;
IF  NOT bTestActiveLiveData THEN
	stStationStruct.nState := 1280;
END_IF


1280: // JOB PASS / JOB FAIL
IF bJobPass  THEN
	GVL_MASTER.stNest.bLeakPass := TRUE;
	GVL_MASTER.stNest.sLeakHMI 	:= "Pass";
	GVL_MASTER.stNest.bLeakReject := FALSE;
   	stStationStruct.nState := 1900;
ELSIF bJobFailed  THEN
   stStationStruct.nState := 1900;
   GVL_MASTER.stNest.bLeakPass := FALSE;
   GVL_MASTER.stNest.sLeakHMI 	:= "Fail";
   GVL_MASTER.stNest.bLeakReject := TRUE;
END_IF

1900:
IF (tonCaseDelay[4].Q AND NOT stStationStruct.bStationManualRequestHMI) OR stStationStruct.bNoCycleStopRequest THEN
	stStationStruct.nState := 1000;
ELSIF tonCaseDelay[4].Q AND stStationStruct.bStationManualRequestHMI THEN
	stStationStruct.nState := 4000;
ELSIF stStationStruct.bStationAbort AND tonCaseDelay[2].Q THEN
	stStationStruct.nState := 100;

END_IF
//=== Manual Mode ===
4000:
IF NOT stStationStruct.bStationManualRequestHMI AND NOT GVL_MASTER.bManualModeTrigger THEN
	stStationStruct.nState := 1000;
ELSIF stStationStruct.bStationAbort THEN
	   stStationStruct.nState := 100;	
END_IF
IF GVL_HMI_GLOBAL.bStartLeakMan THEN
	
	bStart 						:= TRUE;
ELSIF GVL_HMI_GLOBAL.bStopLeakMan THEN
	
	bStop						:= TRUE;

ELSE 
	bStart						:= FALSE;
	bStop						:= FALSE;
END_IF
ACT_ChangeJOB();

9000:

bClearErrorIns 					:= FALSE;
bStart							:= FALSE;
GVL_MASTER.stNest.bLeakPass 	:= FALSE;


stStationStruct.nState := 9100;	
9100:
IF tonCaseDelay[5].Q THEN
	stStationStruct.nState := 9200;
END_IF
9200:
bClearErrorIns := TRUE;
IF tonCaseDelay[6].Q THEN
	stStationStruct.nState := 9300;
END_IF
9300: 
IF bLeakTesterNoError THEN
   stStationStruct.nState := 1000;
END_IF

	
END_CASE

IF NOT bLeakTesterNoError AND NOT stStationStruct.nState >= 9000 THEN
stStationStruct.nState := 9000;
END_IF

ACTION ACT_ChangeJob:
	
GVL_IO.dw_B07_i28General_I_O.bSetProgram[0] := GVL_HMI_GLOBAL.uNewLeakProgID.0;
GVL_IO.dw_B07_i28General_I_O.bSetProgram[1] := GVL_HMI_GLOBAL.uNewLeakProgID.1;
GVL_IO.dw_B07_i28General_I_O.bSetProgram[2] := GVL_HMI_GLOBAL.uNewLeakProgID.2;
GVL_IO.dw_B07_i28General_I_O.bSetProgram[3] := GVL_HMI_GLOBAL.uNewLeakProgID.3;
GVL_IO.dw_B07_i28General_I_O.bSetProgram[4] := GVL_HMI_GLOBAL.uNewLeakProgID.4;
GVL_IO.dw_B07_i28General_I_O.bSetProgram[5] := GVL_HMI_GLOBAL.uNewLeakProgID.5;
GVL_IO.dw_B07_i28General_I_O.bSetProgram[6] := GVL_HMI_GLOBAL.uNewLeakProgID.6;
GVL_IO.dw_B07_i28General_I_O.bSetProgram[7] := GVL_HMI_GLOBAL.uNewLeakProgID.7;


IF GVL_HMI_GLOBAL.bSetLeakProgramID THEN 
	
		uSetProgramID := GVL_HMI_GLOBAL.uNewLeakProgID;
END_IF
END_ACTION

ACTION ACT_IOLINK:


bLeakTesterNoError				:= NOT GVL_IO.dw_B07_i28General_I_O.bMalfunction;
uCurrentProgramID				:= GVL_IO.dw_B07_i28General_I_O.nCurrentProgramNumber;
bProgramAccepted				:= GVL_IO.dw_B07_i28General_I_O.bProgramAccept;
bInstrumentReady				:= GVL_IO.dw_B07_i28General_I_O.bInstrumentReady;
bProgramRejected				:= GVL_IO.dw_B07_i28General_I_O.bProgramReject;
bTestActiveLiveData				:= GVL_IO.dw_B07_i28General_I_O.bTestActiveLiveData;
nLiveMeasID						:= GVL_IO.dw_B07_i28LiveMeasurement.inUniqueID;
nLastMeasID						:= GVL_IO.dw_B07_i28LastResult.inUniqueID;
bJobPass						:= GVL_IO.dw_B07_i28General_I_O.bProgramAccept;
bJobFailed						:= GVL_IO.dw_B07_i28General_I_O.bProgramReject;



GVL_IO.dw_B07_i28General_I_O.bStart 			:= bStart;
GVL_IO.dw_B07_i28General_I_O.bStop				:= bStop OR stStationStruct.bStationAbort;
GVL_IO.dw_B07_i28General_I_O.bChangeProgram := GVL_HMI_GLOBAL.bSetLeakProgramID;
GVL_IO.dw_B07_i28General_I_O.bReset := bClearErrorIns OR GVL_HMI_GLOBAL.bResetLeakMan;



GVL_HMI_GLOBAL.nLeakTestCycTime := (TIME_TO_DINT(GVL_MASTER.stAlarms[1].aEventTimers[1].ET))/1000;

IF GVL_IO.dw_B07_i28LiveMeasurement.inMeasurement2 <> 0 THEN 
rPressure:=UDINT_TO_REAL(GVL_IO.dw_B07_i28LiveMeasurement.inMeasurement2);
END_IF
END_ACTION

ACTION ACT_TimTrig:


tonCaseDelay[1](IN:= (stStationStruct.nState=400),PT:=T#50MS);
tonCaseDelay[2](IN:= (stStationStruct.nState=160),PT:=T#50MS);
tonCaseDelay[3](IN:= (stStationStruct.nState=1200),PT:=T#5S);
tonCaseDelay[4](IN:= (stStationStruct.nState=1900),PT:=T#1S);
tonCaseDelay[5](IN:= (stStationStruct.nState=9100),PT:=T#200MS);
tonCaseDelay[6](IN:= (stStationStruct.nState=9200),PT:=T#250MS);
tonCaseDelay[7](IN:= ,PT:=T#500MS);



rtrigCaseTriger[1](clk:= (stStationStruct.nState=1900) AND bJobPass);
rtrigCaseTriger[2](clk:= (stStationStruct.nState=1900) AND bJobFailed);
rtrigCaseTriger[3](clk:= stStationStruct.bStationAbort);
END_ACTION

END_PROGRAM

// ---- POUs/A_Master/PRG_MachineStatus.TcPOU
PROGRAM PRG_MachineStatus
VAR

	tonPowerUp						: TON;
	tonSystemInitialising			: TON;
	tonSystemInitialisingTimeout	: TON;
	
	bMemoSystemReadyToStart			:BOOL; //flag set only once to establissh if system was in ready to start state after powerUP
	
// =========== Manual =============	

	rtrigManualModeOFF              :ARRAY[1..4] OF R_TRIG;
	rtrigManualMode                 :R_TRIG;	
		// =========== Master Time =============
		//Variables
	bReadyToRead				:BOOL;
	bFirstScan					:BOOL := TRUE;
	bUpdateSysTime				:BOOL; //Output of pulse generator
	tSysTimeUpdatePeriod		:TIME := T#5S;
	stTimeStamp					:TIMESTRUCT;
	stNullTimeStamp				:TIMESTRUCT;
	sRawDateTime				:STRING;

	

	
	
	sDateTime					:STRING;
	sDateTimeSpaces				:STRING;
	
	
	
	//Functions
	fbGetSystemTime				:TC2_Utilities.NT_GetTime;
	fbRTClock					:TC2_Utilities.RTC_EX2;		//Local real-time clock
	tonTimeUpdateGen			:TC2_Utilities.TON;			//Pulse generator for triggering fbGetSystemTime function
	rtrigSysTimeCollected		:TC2_Utilities.R_TRIG;		//System time collected



		
END_VAR

ACT_ManualMode();
ACT_MasterTime();
ACT_MachineStatusBaner();


(*Power Up*)

tonPowerUp( IN := TRUE,  PT := T#5S, Q => GVL_MASTER.stMasterControl.bPowerUpTimerComplete );

(*System Initialising*)

tonSystemInitialising( IN := (GVL_MASTER.stMachineStatus.eMachineState = E_MachineState.SYSTEM_INITIALISING),
	PT := T#1S,
	Q => GVL_MASTER.stMasterControl.bSystemInitialisingTimerComplete);
	
(*System Initialising Timeout*)
	
tonSystemInitialisingTimeout(IN := (GVL_MASTER.stMachineStatus.eMachineState = E_MachineState.SYSTEM_INITIALISING),
	PT := T#5M,
	Q => GVL_MASTER.stMasterControl.bSystemInitialisingTimeoutComplete);
	
(* Set Machine State to Power Up while waiting for Power Up Timer to Complete *)
IF NOT GVL_MASTER.stMasterControl.bPowerUpTimerComplete THEN
	GVL_MASTER.stMachineStatus.eMachineState := E_MachineState.SYSTEM_POWER_UP;
END_IF

(********************************(Sequence )*******************************************************)
(* Move to Immediate Stopped once there is an Immediate Fault *)
IF NOT GVL_MASTER.stMasterControl.bNoMachineImmediateFault THEN		
	GVL_MASTER.stMachineStatus.eMachineState := E_MachineState.IMMEDIATE_STOPPED;
ELSIF NOT GVL_MASTER.stMasterControl.bNoCycleStopFault THEN
	GVL_MASTER.stMachineStatus.eMachineState := E_MachineState.CYCLE_STOP_FAULT;	
END_IF

CASE GVL_MASTER.stMachineStatus.eMachineState OF
	
E_MachineState.SYSTEM_POWER_UP:
	
	bMemoSystemReadyToStart:=FALSE;
	(* Move to Immediate Stopped once Power Up Timer has completed *)
	IF GVL_MASTER.stMasterControl.bPowerUpTimerComplete THEN			
		GVL_MASTER.stMachineStatus.eMachineState := E_MachineState.IMMEDIATE_STOPPED;
	END_IF
	
E_MachineState.IMMEDIATE_STOPPED:	
	(* Move to System Initialising once there is no Immediate Fault *)
	IF GVL_MASTER.stMasterControl.bNoMachineImmediateFault  THEN	
		GVL_MASTER.stMachineStatus.eMachineState := E_MachineState.SYSTEM_INITIALISING;
	(* Move to Immediate Fault once there is an Immediate Fault *)
	ELSIF NOT GVL_MASTER.stMasterControl.bNoMachineImmediateFault THEN
		GVL_MASTER.stMachineStatus.eMachineState := E_MachineState.IMMEDIATE_FAULT;	
	END_IF
	
E_MachineState.SYSTEM_INITIALISING:		
	IF  GVL_MASTER.stMasterControl.bNoMachineImmediateFault	 AND GVL_MASTER.stMasterControl.bSystemInitialisingTimerComplete  THEN		
		GVL_MASTER.stMachineStatus.eMachineState := E_MachineState.SYSTEM_READY_TO_START;
	
	//Move to Cycle Stopped once there is a Cycle Stop Request AND All Stations are Cycle Stopped AND there is No Immediate Fault*)
	ELSIF GVL_HMI_GLOBAL.bStopButton
		OR (GVL_MASTER.stMasterControl.bNoMachineImmediateFault 
		AND (GVL_MASTER.stMasterControl.bSystemInitialisingTimeoutComplete OR GVL_MASTER.stMasterControl.bCycleStopRequest) AND GVL_MASTER.stMasterControl.bAllStationsCycledStopped)
	THEN		
		GVL_MASTER.stMachineStatus.eMachineState := E_MachineState.CYCLE_STOPPED;			
	ELSIF GVL_MASTER.stMasterControl.bNoMachineImmediateFault AND NOT GVL_MASTER.stMasterControl.bNoCycleStopFault THEN		
		GVL_MASTER.stMachineStatus.eMachineState := E_MachineState.CYCLE_STOP_FAULT;	
	ELSIF NOT GVL_MASTER.stMasterControl.bNoStationImmediateFault THEN
         GVL_MASTER.stMachineStatus.eMachineState := E_MachineState.IMMEDIATE_FAULT;
      	
	END_IF
	
E_MachineState.SYSTEM_READY_TO_START:
	bMemoSystemReadyToStart := TRUE;
	
	//Move to System Auto if the Start Button has been pressed
	IF GVL_MASTER.stMasterControl.bManualModeRequest THEN
		GVL_MASTER.stMachineStatus.eMachineState := E_MachineState.MANUAL_MODE;
	
	ELSIF GVL_HMI_GLOBAL.bStopButton THEN
        GVL_MASTER.stMachineStatus.eMachineState := E_MachineState.STOPPING; 
	ELSIF GVL_HMI_GLOBAL.bStartButton AND NOT PRG_Mastercycle.biClamp AND NOT PRG_Mastercycle.biPartPresent    THEN		//**LA 12092025	
		GVL_MASTER.stMachineStatus.eMachineState := E_MachineState.SYSTEM_AUTO_CYCLE;
		
	//Move to Cycle Stopped once there is a Cycle Stop Request AND All Stations are Cycle Stopped AND there is No Immediate Fault
	ELSIF (GVL_MASTER.stMasterControl.bCycleStopRequest OR NOT	GVL_MASTER.stMasterControl.bNoCycleStopFault) 
	AND GVL_MASTER.stMasterControl.bNoMachineImmediateFault
	THEN				
		GVL_MASTER.stMachineStatus.eMachineState := E_MachineState.CYCLE_STOPPED;	
	ELSIF NOT GVL_MASTER.stMasterControl.bNoCycleStopFault THEN
		GVL_MASTER.stMachineStatus.eMachineState := E_MachineState.CYCLE_STOP_FAULT;
	ELSIF NOT GVL_MASTER.stMasterControl.bNoMachineImmediateFault OR NOT GVL_MASTER.stMasterControl.bNoStationImmediateFault THEN
       GVL_MASTER.stMachineStatus.eMachineState := E_MachineState.IMMEDIATE_FAULT ;	
	   
	END_IF
	

	
	
	
E_MachineState.SYSTEM_AUTO_CYCLE:	
	//Move to System Dwell once there is a Dwell Request
	IF GVL_MASTER.stMasterControl.bDwellRequest THEN
		GVL_MASTER.stMachineStatus.eMachineState := E_MachineState.SYSTEM_DWELL;
	
	//Move to Cycle Stopped once there is a Cycle Stop Request AND All Stations are Cycle Stopped AND there is No Immediate Fault OR when cycle done
	ELSIF NOT GVL_MASTER.stMasterControl.bNoCycleStopFault THEN //Fast cycle stop	
		GVL_MASTER.stMachineStatus.eMachineState := E_MachineState.CYCLE_STOP_FAULT;
	(*ELSIF GVL_Master.bMachineCycleDone   THEN 
	stMachineStatus.eMachineState := E_MachineState.CYCLE_STOPPED; //Instant cycle stop???		*)
	ELSIF GVL_HMI_GLOBAL.bStopButton OR GVL_MASTER.stMasterControl.bCycleStopRequest OR GVL_HMI_GLOBAL.nRegionMain <> 1 THEN
		GVL_MASTER.stMachineStatus.eMachineState := E_MachineState.STOPPING; //Stopping sequence 
	ELSIF NOT GVL_MASTER.stMasterControl.bNoStationImmediateFault OR NOT GVL_MASTER.stMasterControl.bNoMachineImmediateFault THEN
     	GVL_MASTER.stMachineStatus.eMachineState := E_MachineState.IMMEDIATE_FAULT;
	END_IF	
	
E_MachineState.SYSTEM_DWELL:		
	(* Move to System Auto Cycle once the Start Button is Pressed AND there is No Dwell Request *)
	IF NOT GVL_MASTER.stMasterControl.bDwellRequest THEN
		GVL_MASTER.stMachineStatus.eMachineState := E_MachineState.SYSTEM_AUTO_CYCLE;	
	(* Move to Cycle Stopped once there is a Cycle Stop Request AND All Stations are Cycle Stopped AND there is No Immediate Fault*)
	ELSIF (GVL_MASTER.stMasterControl.bCycleStopRequest OR	NOT	GVL_MASTER.stMasterControl.bNoCycleStopFault) 
		AND GVL_MASTER.stMasterControl.bAllStationsCycledStopped AND GVL_MASTER.stMasterControl.bNoMachineImmediateFault
	THEN				
		GVL_MASTER.stMachineStatus.eMachineState := E_MachineState.CYCLE_STOPPED;	
	END_IF

E_MachineState.STOPPING: 
	IF  GVL_MASTER.stMasterControl.bAllStationsCycledStopped THEN
		GVL_MASTER.stMachineStatus.eMachineState := E_MachineState.CYCLE_STOPPED;
	ELSIF NOT GVL_MASTER.stMasterControl.bNoCycleStopFault THEN
		GVL_MASTER.stMachineStatus.eMachineState := E_MachineState.CYCLE_STOP_FAULT;
	ELSIF NOT GVL_MASTER.stMasterControl.bNoMachineImmediateFault OR NOT GVL_MASTER.stMasterControl.bNoStationImmediateFault THEN
        GVL_MASTER.stMachineStatus.eMachineState := E_MachineState.IMMEDIATE_FAULT ;
	END_IF
	
E_MachineState.CYCLE_STOPPED:
	IF GVL_MASTER.stMasterControl.bManualModeRequest THEN
		GVL_MASTER.stMachineStatus.eMachineState := E_MachineState.MANUAL_MODE;			
	(* Move to System Initialising once there is no Cycle Stop Fault AND the Reset Button is Pressed *)
	ELSIF (GVL_MASTER.stMasterControl.bNoCycleStopFault AND GVL_HMI_GLOBAL.bResetButton )THEN
		GVL_MASTER.stMachineStatus.eMachineState := E_MachineState.SYSTEM_INITIALISING;		
	ELSIF NOT GVL_MASTER.stMasterControl.bNoStationImmediateFault THEN
       	GVL_MASTER.stMachineStatus.eMachineState := E_MachineState.IMMEDIATE_FAULT;
	END_IF	

E_MachineState.CYCLE_STOP_FAULT:	
	(* Move to Cycle Stopped once there no Cycle Stop Fault AND there is No Immediate Fault*)
	IF GVL_MASTER.stMasterControl.bNoCycleStopFault THEN
		GVL_MASTER.stMachineStatus.eMachineState := E_MachineState.CYCLE_STOPPED;
	END_IF	
ELSE 	
	GVL_MASTER.stMachineStatus.eMachineState := E_MachineState.SYSTEM_POWER_UP;	
	
E_MachineState.MANUAL_MODE:

	IF NOT GVL_MASTER.stMasterControl.bManualModeRequest THEN
		GVL_MASTER.stMachineStatus.eMachineState := E_MachineState.CYCLE_STOPPED;
	END_IF
	
E_MachineState.IMMEDIATE_FAULT:		
	(* Move to Immediate Stopped once there is an Immediate Fault *)
	IF GVL_MASTER.stMasterControl.bNoMachineImmediateFault AND  GVL_MASTER.stMasterControl.bNoStationImmediateFault THEN
		GVL_MASTER.stMachineStatus.eMachineState := E_MachineState.IMMEDIATE_STOPPED;		

	END_IF
END_CASE
//////////////////////////////////////////////////////////////////////////////////////////////////////////////
								//CYCLE STOP REQUEST//
//////////////////////////////////////////////////////////////////////////////////////////////////////////////
IF GVL_MASTER.stAlarms[0].bCycleStopRequest OR GVL_MASTER.stAlarms[1].bCycleStopRequest  THEN
				GVL_MASTER.stMasterControl.bCycleStopRequest	:=	TRUE;
ELSE			GVL_MASTER.stMasterControl.bCycleStopRequest	:=	FALSE;
END_IF




(************************************* write all system states to variables ***********************)

GVL_MASTER.stMachineStatus.bSystemPowerUp :=(GVL_MASTER.stMachineStatus.eMachineState = E_MachineState.SYSTEM_POWER_UP);
GVL_MASTER.stMachineStatus.bImmediateStopped :=(GVL_MASTER.stMachineStatus.eMachineState = E_MachineState.IMMEDIATE_STOPPED);
GVL_MASTER.stMachineStatus.bSystemInitialising :=(GVL_MASTER.stMachineStatus.eMachineState = E_MachineState.SYSTEM_INITIALISING);
GVL_MASTER.stMachineStatus.bSystemReadyToStart := (GVL_MASTER.stMachineStatus.eMachineState = E_MachineState.SYSTEM_READY_TO_START);
GVL_MASTER.stMachineStatus.bSystemAutoCycle := (GVL_MASTER.stMachineStatus.eMachineState = E_MachineState.SYSTEM_AUTO_CYCLE);
GVL_MASTER.stMachineStatus.bSystemDwell := (GVL_MASTER.stMachineStatus.eMachineState = E_MachineState.SYSTEM_DWELL);
GVL_MASTER.stMachineStatus.bSystemStopping := (GVL_MASTER.stMachineStatus.eMachineState = E_MachineState.STOPPING);
GVL_MASTER.stMachineStatus.bCycleStopped := (GVL_MASTER.stMachineStatus.eMachineState = E_MachineState.CYCLE_STOPPED);
GVL_MASTER.stMachineStatus.bManualMode := (GVL_MASTER.stMachineStatus.eMachineState = E_MachineState.MANUAL_MODE);
GVL_MASTER.stMachineStatus.bImmediateFault := (GVL_MASTER.stMachineStatus.eMachineState = E_MachineState.IMMEDIATE_FAULT);
GVL_MASTER.stMachineStatus.bCycleStopFault := (GVL_MASTER.stMachineStatus.eMachineState = E_MachineState.CYCLE_STOP_FAULT);

ACTION ACT_MachineStatusBaner:
//Machine status banner action
//SYSTEM POWER UP
IF GVL_MASTER.stMachineStatus.bSystemPowerUp THEN	
	GVL_MASTER.stMachineStatus.sMachineStatusText := 'SYSTEM POWER UP';		// fill colour WHITE, text colour BLACK
	GVL_MASTER.stMachineStatus.nMachineStatusColour := nWHITE;
	GVL_MASTER.stMachineStatus.nMachineStatusTxtCol := nBLACK;
	GVL_MASTER.stMachineStatus.sBannerBckColor := sWHITE;
	GVL_MASTER.stMachineStatus.sBannerTextColor := sBLACK;
END_IF

(* IMMEDIATE STOPPED *)
IF GVL_MASTER.stMachineStatus.bImmediateStopped THEN	
	GVL_MASTER.stMachineStatus.sMachineStatusText := 'IMMEDIATE STOPPED';		// fill colour BLACK, text colour WHITE
	GVL_MASTER.stMachineStatus.nMachineStatusColour := nBLACK;
	GVL_MASTER.stMachineStatus.nMachineStatusTxtCol := nWHITE;
	GVL_MASTER.stMachineStatus.sBannerBckColor := sBLACK;
	GVL_MASTER.stMachineStatus.sBannerTextColor := sWHITE;	
END_IF

(* SYSTEM INITIALISING *)
IF GVL_MASTER.stMachineStatus.bSystemInitialising THEN	
	GVL_MASTER.stMachineStatus.sMachineStatusText := 'SYSTEM INITIALIZING';		// fill colour YELLOW, text colour BLACK
	GVL_MASTER.stMachineStatus.nMachineStatusColour := nYELLOW;
	GVL_MASTER.stMachineStatus.nMachineStatusTxtCol := nBLACK;
	GVL_MASTER.stMachineStatus.sBannerBckColor := sYELLOW;
	GVL_MASTER.stMachineStatus.sBannerTextColor := sBLACK;
END_IF
(*
(* SYSTEM IN STANDBY *)
IF stMachineStatus.bSystemStandby THEN
	stMachineStatus.sMachineStatusText := 'SYSTEM IN STANDBY';
	stMachineStatus.nMachineStatusColour := nORANGE;
	stMachineStatus.nMachineStatusTxtCol := nWHITE;
END_IF
*)
(* SYSTEM READY TO START FLASH ON *)
IF GVL_MASTER.stMachineStatus.bSystemReadyToStart AND GVL_MASTER.bFlash1Hz THEN
	GVL_MASTER.stMachineStatus.sMachineStatusText := 'SYSTEM READY TO START';		// fill colour GREEN, text colour WHITE
	GVL_MASTER.stMachineStatus.nMachineStatusColour := nGREEN;
	GVL_MASTER.stMachineStatus.nMachineStatusTxtCol := nWHITE;
	GVL_MASTER.stMachineStatus.sBannerBckColor := sGREEN;
	GVL_MASTER.stMachineStatus.sBannerTextColor := sWHITE;
END_IF

(* SYSTEM READY TO START FLASH OFF *)
IF GVL_MASTER.stMachineStatus.bSystemReadyToStart AND NOT GVL_MASTER.bFlash1Hz THEN	
	GVL_MASTER.stMachineStatus.sMachineStatusText := 'SYSTEM READY TO START';		// fill colour WHITE, text colour GREEN
	GVL_MASTER.stMachineStatus.nMachineStatusColour := nWHITE;
	GVL_MASTER.stMachineStatus.nMachineStatusTxtCol := nGREEN;
	GVL_MASTER.stMachineStatus.sBannerBckColor := sWHITE;
	GVL_MASTER.stMachineStatus.sBannerTextColor := sGREEN;
END_IF

(* SYSTEM AUTO CYCLE *)
IF GVL_MASTER.stMachineStatus.bSystemAutoCycle THEN	
	GVL_MASTER.stMachineStatus.sMachineStatusText := 'SYSTEM AUTO CYCLE';		// fill colour GREEN, text colour WHITE
	GVL_MASTER.stMachineStatus.nMachineStatusColour := nGREEN;
	GVL_MASTER.stMachineStatus.nMachineStatusTxtCol := nWHITE;
	GVL_MASTER.stMachineStatus.sBannerBckColor := sGREEN;
	GVL_MASTER.stMachineStatus.sBannerTextColor := sWHITE;	
END_IF

(* SYSTEM DWELL *)
IF GVL_MASTER.stMachineStatus.bSystemDwell THEN	
	GVL_MASTER.stMachineStatus.sMachineStatusText := 'SYSTEM DWELL';		// fill colour ORANGE, text colourWHITE
	GVL_MASTER.stMachineStatus.nMachineStatusColour := nORANGE;
	GVL_MASTER.stMachineStatus.nMachineStatusTxtCol := nWHITE;
	GVL_MASTER.stMachineStatus.sBannerBckColor := sORANGE;
	GVL_MASTER.stMachineStatus.sBannerTextColor := sWHITE;	
END_IF

(* STOPPING *)
IF GVL_MASTER.stMachineStatus.bSystemStopping AND GVL_MASTER.bFlash1Hz THEN	
	GVL_MASTER.stMachineStatus.sMachineStatusText := 'STOPPING';		// fill colour BLACK, text colour WHITE
	GVL_MASTER.stMachineStatus.nMachineStatusColour := nBLACK;
	GVL_MASTER.stMachineStatus.nMachineStatusTxtCol := nWHITE;
	GVL_MASTER.stMachineStatus.sBannerBckColor := sBLACK;
	GVL_MASTER.stMachineStatus.sBannerTextColor := sWHITE;	
END_IF

(* STOPPING *)
IF GVL_MASTER.stMachineStatus.bSystemStopping AND NOT GVL_MASTER.bFlash1Hz THEN	
	GVL_MASTER.stMachineStatus.sMachineStatusText := 'STOPPING';		// fill colour WHITE, text colour BLACK
	GVL_MASTER.stMachineStatus.nMachineStatusColour := nWHITE;
	GVL_MASTER.stMachineStatus.nMachineStatusTxtCol := nBLACK;
	GVL_MASTER.stMachineStatus.sBannerBckColor := sWHITE;
	GVL_MASTER.stMachineStatus.sBannerTextColor := sBLACK;	
END_IF

(* CYCLE STOPPED *)
IF GVL_MASTER.stMachineStatus.bCycleStopped THEN	
	GVL_MASTER.stMachineStatus.sMachineStatusText := 'CYCLE STOPPED';		// fill colour BLACK, text colour WHITE
	GVL_MASTER.stMachineStatus.nMachineStatusColour := nBLACK;
	GVL_MASTER.stMachineStatus.nMachineStatusTxtCol := nWHITE;
	GVL_MASTER.stMachineStatus.sBannerBckColor := sBLACK;
	GVL_MASTER.stMachineStatus.sBannerTextColor := sWHITE;	
END_IF

(* IMMEDIATE FAULT FLASH ON *)
IF GVL_MASTER.stMachineStatus.bImmediateFault AND GVL_MASTER.bFlash1Hz THEN	
	GVL_MASTER.stMachineStatus.sMachineStatusText := 'IMMEDIATE FAULT';		// fill colour RED, text colour WHITE
	GVL_MASTER.stMachineStatus.nMachineStatusColour := nRED;
	GVL_MASTER.stMachineStatus.nMachineStatusTxtCol := nWHITE;
	GVL_MASTER.stMachineStatus.sBannerBckColor := sRED;
	GVL_MASTER.stMachineStatus.sBannerTextColor := sWHITE;	
END_IF

(* IMMEDIATE FAULT FLASH OFF *)
IF GVL_MASTER.stMachineStatus.bImmediateFault AND NOT GVL_MASTER.bFlash1Hz THEN	
	GVL_MASTER.stMachineStatus.sMachineStatusText := 'IMMEDIATE FAULT';		// fill colour WHITE, text colour BLACK
	GVL_MASTER.stMachineStatus.nMachineStatusColour := nWHITE;
	GVL_MASTER.stMachineStatus.nMachineStatusTxtCol := nBLACK;
	GVL_MASTER.stMachineStatus.sBannerBckColor := sWHITE;
	GVL_MASTER.stMachineStatus.sBannerTextColor := sBLACK;	
END_IF

(* CYCLE STOP FAULT FLASH ON *)
IF GVL_MASTER.stMachineStatus.bCycleStopFault AND GVL_MASTER.bFlash1Hz THEN	
	GVL_MASTER.stMachineStatus.sMachineStatusText := 'CYCLE STOP FAULT';		// fill colour RED, text colour WHITE
	GVL_MASTER.stMachineStatus.nMachineStatusColour := nRED;
	GVL_MASTER.stMachineStatus.nMachineStatusTxtCol := nWHITE;
	GVL_MASTER.stMachineStatus.sBannerBckColor := sRED;
	GVL_MASTER.stMachineStatus.sBannerTextColor := sWHITE;	
END_IF

(* CYCLE STOP FAULT FLASH OFF *)
IF GVL_MASTER.stMachineStatus.bCycleStopFault AND NOT GVL_MASTER.bFlash1Hz THEN	
	GVL_MASTER.stMachineStatus.sMachineStatusText := 'CYCLE STOP FAULT';		// fill colour WHITE, text colour RED
	GVL_MASTER.stMachineStatus.nMachineStatusColour := nWHITE;
	GVL_MASTER.stMachineStatus.nMachineStatusTxtCol := nRED;
	GVL_MASTER.stMachineStatus.sBannerBckColor := sWHITE;
	GVL_MASTER.stMachineStatus.sBannerTextColor := sRED;	
END_IF

(* MANUAL MODE *)
IF GVL_MASTER.stMachineStatus.bManualMode THEN	
	GVL_MASTER.stMachineStatus.sMachineStatusText := 'MANUAL MODE';		// fill colour BLUE text colour WHITE
	GVL_MASTER.stMachineStatus.nMachineStatusColour := nBLUE;
	GVL_MASTER.stMachineStatus.nMachineStatusTxtCol := nWHITE;
	GVL_MASTER.stMachineStatus.sBannerBckColor := sBLUE;
	GVL_MASTER.stMachineStatus.sBannerTextColor := sWHITE;	
END_IF

(*
(* SYSTEM READY TO START FLASH ON *)
IF stMachineStatus.bSystemPurge AND bFlash1Hz THEN
	stMachineStatus.sMachineStatusText := 'SYSTEM PURGE';		// fill colour GREEN, text colour WHITE
	stMachineStatus.nMachineStatusColour := nORANGE;
	stMachineStatus.nMachineStatusTxtCol := nBLACK;
	stMachineStatus.sBannerBckColor := sORANGE;
	stMachineStatus.sBannerTextColor := sBLACK;	
END_IF

(* SYSTEM READY TO START FLASH OFF *)
IF stMachineStatus.bSystemPurge AND NOT bFlash1Hz THEN	
	stMachineStatus.sMachineStatusText := 'SYSTEM PURGE';		// fill colour WHITE, text colour GREEN
	stMachineStatus.nMachineStatusColour := nWHITE;
	stMachineStatus.nMachineStatusTxtCol := nBLUE;
	stMachineStatus.sBannerBckColor := sWHITE;
	stMachineStatus.sBannerTextColor := sBLUE;	
END_IF
*)
(*
(* CALIBRATION *)
IF stMachineStatus.bCalibrationFlag AND bFlash1Hz THEN	
	stMachineStatus.sMachineStatusText := 'CALIBRATION MODE';		// fill colour BLUE text colour WHITE
	stMachineStatus.nMachineStatusColour := nBLUE;
	stMachineStatus.nMachineStatusTxtCol := nWHITE;
	stMachineStatus.sBannerBckColor := sBLUE;
	stMachineStatus.sBannerTextColor := sWHITE;	
END_IF
IF stMachineStatus.bCalibrationFlag AND NOT bFlash1Hz THEN	
	stMachineStatus.sMachineStatusText := 'CALIBRATION MODE';		// fill colour BLUE text colour WHITE
	stMachineStatus.nMachineStatusColour := nWHITE;
	stMachineStatus.nMachineStatusTxtCol := nBLUE;
	stMachineStatus.sBannerBckColor := sWHITE;
	stMachineStatus.sBannerTextColor := sBLUE;	
END_IF
*)
END_ACTION

ACTION ACT_ManualMode:
IF	 GVL_MASTER.stMachineStatus.bSystemReadyToStart THEN
	GVL_HMI_GLOBAL.bEnableManualMode := TRUE;
ELSE GVL_HMI_GLOBAL.bEnableManualMode := FALSE;
END_IF


rtrigManualMode(CLK:= GVL_HMI_GLOBAL.nRegionMain=10);
rtrigManualModeOFF[1](CLK:=GVL_Master.stMachineStatus.bManualMode AND (GVL_HMI_GLOBAL.nRegionMain <> 10));
rtrigManualModeOFF[2](CLK:=GVL_Master.stMachineStatus.bManualMode AND GVL_HMI_GLOBAL.bStopButton);
rtrigManualModeOFF[3](CLK:=GVL_Master.stMachineStatus.bManualMode AND NOT GVL_Master.stMasterControl.bNoStationImmediateFault );
rtrigManualModeOff[4](CLK := GVL_HMI_GLOBAL.bManualModeOff[1], Q => GVL_HMI_GLOBAL.bManualModeOff[2]);

IF rtrigManualMode.Q THEN 
	GVL_Master.stMasterControl.bManualModeRequest := TRUE;
	GVL_HMI_GLOBAL.bManualModeOff[1] := FALSE;
ELSIF rtrigManualModeOFF[1].Q OR rtrigManualModeOFF[2].Q OR rtrigManualModeOFF[3].Q THEN
	GVL_HMI_GLOBAL.nRegionMain:=1;
	GVL_Master.stMasterControl.bManualModeRequest := FALSE ;
	GVL_HMI_GLOBAL.bManualModeOff[1] := TRUE;
	
	
ELSE GVL_HMI_GLOBAL.bManualModeOff[1] := FALSE;
	
END_IF





IF GVL_Master.stMachineStatus.bManualMode  THEN
	GVL_Master.stStationSruct[1].bStationManualRequestHMI := TRUE;

ELSE
    GVL_Master.stStationSruct[1].bStationManualRequestHMI := FALSE;

END_IF
END_ACTION

ACTION ACT_MasterTime:
//Aux functions call
tonTimeUpdateGen(	IN := NOT bUpdateSysTime,
					PT := tSysTimeUpdatePeriod,
					Q => bUpdateSysTime);

